// TwinCAT 3 PLC project Transport
// ProgramVersion: 3.1.4026.21
// CompilerDefines: VISU_USEPROPERTYINFO
// libraries:
//   Tc2_Standard, * (Beckhoff Automation GmbH)
//   Tc2_System, * (Beckhoff Automation GmbH)
//   VisuDialogs, * (System)
// project tree:
//   001DUTs/ENUM/ E_CmdState.TcDUT, E_ErrorLevel.TcDUT, E_Mode.TcDUT, E_Convoyer.TcDUT, E_LTUPosition.TcDUT, E_RouteStepType.TcDUT, E_SetChild.TcDUT
//   001DUTs/GVL_Base/ GVL_Core.TcGVL
//   001DUTs/ITF/Device/ ITF_Convoyer.TcIO, ITF_LTU.TcIO, ITF_RouteProvider.TcIO
//   001DUTs/ITF/Generic/ ITF_Base.TcIO, ITF_Device.TcIO
//   001DUTs/ITF/ ITF_Owner.TcIO
//   001DUTs/STRUCT/ ST_ErrorInfo.TcDUT, ST_MaschineHMI.TcDUT, ST_Route.TcDUT, ST_RouteJob.TcDUT, ST_RouteStep.TcDUT
//   002 POUs/00 Generic/ FD_Device.TcPOU, FB_Base.TcPOU, FM_Maschine.TcPOU
//   002 POUs/01 Lib/01 Device/00 Template/ FB_Template.TcPOU (not stored)
//   002 POUs/01 Lib/01 Device/ FD_RouteManagerDevice.TcPOU, FD_LUTDevice.TcPOU (not stored), FD_ConvoyerDevice.TcPOU, FD_RouteExecutorDevice.TcPOU
//   002 POUs/01 Lib/02 SimpleDevice/00 Template/ FB_TemplateSimpleDevice.TcPOU
//   002 POUs/01 Lib/02 SimpleDevice/ FB_ReadHead.TcPOU, FB_PneuCyl_Stopper.TcPOU, FB_SimpleMotor.TcPOU (not stored), FB_PneuCyl_3Pos.TcPOU
//   002 POUs/01 Lib/Digit I_O/Input/ FB_Input.TcPOU (not stored)
//   002 POUs/01 Lib/Digit I_O/Output/ FB_Output.TcPOU
//   1000 Maschine xxx/01 DUTs/GVLs/ GVL_Customer.TcGVL
//   1000 Maschine xxx/01 DUTs/STRUCT/ ST_HmiCustomer.TcDUT
//   1000 Maschine xxx/ MAIN.TcPOU
//   1000 Maschine xxx/_Customer/ FM_Customer.TcPOU
//   1000 Maschine xxx/_Customer/VISUs/ Visu_Customer.TcVIS
//   / GlobalTextList.TcGTLO, PlcTask.TcTTO, Visualisierungsmanager.TcVMO (not stored)
// real-time tasks:
//   TASK PlcTask: cycle T#10ms, priority 20, ADS port 350

CONFIGURATION Transport
    RESOURCE PLC ON TwinCAT3
        TASK PlcTask(INTERVAL := T#10ms, PRIORITY := 20);
        PROGRAM MAIN WITH PlcTask : MAIN;
    END_RESOURCE
END_CONFIGURATION

// ---- 001DUTs/ENUM/E_CmdState.TcDUT

{attribute 'qualified_only'}
{attribute 'strict'}
{attribute 'to_string'}

(*

*)
TYPE E_CmdState :
(
	//====================  
	//											
	Idle							:=  0,
	Succeeded 				:=  1,
	Error	    				:=  2,
	Timeout						:=  3,
	Aborted	    			:=  4,
	Deleted						:=  5,
	Reseted						:=  6,
	NotReady					:=  7,
	Failed						:=  8,
	Hold							:=  9,
	
	//==================== 
	Busy							:= 15
);
END_TYPE

// ---- 001DUTs/ENUM/E_ErrorLevel.TcDUT

{attribute 'qualified_only'}
{attribute 'strict'}
{attribute 'to_string'}
TYPE E_ErrorLevel :
(
	NONE := 0,
	Low,
	High,
	Critical
)UINT;
END_TYPE

// ---- 001DUTs/ENUM/E_Mode.TcDUT
{attribute 'qualified_only'}
{attribute 'strict'}
{attribute 'to_string'}
TYPE E_Mode :
(
 	Idle := 0,
 	Homing,
 	Service,
 	Auto,
 	Error
)UINT;
END_TYPE

// ---- 001DUTs/ENUM/E_Convoyer.TcDUT
{attribute 'qualified_only'}
{attribute 'strict'}
{attribute 'to_string'}
(*

*)
TYPE E_Convoyer :
(
	Convoyer_NONE := 0,
  Convoyer_3		:=3,
  Convoyer_6		:=6,
  Convoyer_9		:=9,
  Convoyer_12		:=12
)UINT;
END_TYPE

// ---- 001DUTs/ENUM/E_LTUPosition.TcDUT
{attribute 'qualified_only'}
{attribute 'strict'}
{attribute 'to_string'}

(*
	Used to define:
	Current LTU position
	Target position (position cible)
	Routing steps
*)

TYPE E_LTUPosition :
(
 	LTU_Unknown := 0,
  LTU_Bottom,
  LTU_Middle,
  LTU_Top
)UINT;
END_TYPE

// ---- 001DUTs/ENUM/E_RouteStepType.TcDUT
{attribute 'qualified_only'}
{attribute 'strict'}
{attribute 'to_string'}
(*
	this ENUM describes elementary actions the system
*)
TYPE E_RouteStepType :
(
 	Route_NONE := 0,

  Route_SetLTUPosition,
  Route_StartConveyor,
  Route_StopConveyor,
  
  Route_StartLTUMotor,
  Route_StopLTUMotor,
  
  Route_WaitLTUOccupied,
  Route_WaitLTUFree,
  Route_WaitLTUPosition,
  
  Route_OpenStopper,
  Route_CloseStopper
)UINT;
END_TYPE

// ---- 001DUTs/ENUM/E_SetChild.TcDUT

{attribute 'qualified_only'}
TYPE E_SetChild :
(
	None					:= 0,
	Enable				:= 1,
	Reset  				:= 3,
	Abort 				:= 4,
	ClearError  	:= 5,
	EStop			  	:= 6,
	Auto  			  := 7,
	Servic				:= 8,
	Home 					:= 9,
	Release		  	:= 10
);
END_TYPE

// ---- 001DUTs/STRUCT/ST_ErrorInfo.TcDUT

TYPE ST_ErrorInfo :
STRUCT
	bActive       : BOOL;
	uiErrorID     : UINT;
	eLevel        : E_ErrorLevel;
	
	sOwner        : STRING(80);
	sMessage      : STRING(255);
	sFullMessage  : STRING(255);
END_STRUCT
END_TYPE

// ---- 001DUTs/STRUCT/ST_MaschineHMI.TcDUT
TYPE ST_MaschineHMI :
STRUCT
	// Commands from HMI
	bCmdHome     					: BOOL;
	bCmdAuto     					: BOOL;
	bCmdService  					: BOOL;
	bCmdStop     					: BOOL;
	bCmdReset    					: BOOL;
	bCmdAbort    					: BOOL;
	
	// Status to HMI
	bEnabled     					: BOOL;
	bReady       					: BOOL;
	bHomed       					: BOOL;
	bBusy        					: BOOL;
	bDone        					: BOOL;
	bError       					: BOOL;
	             					
	eMode        					: E_Mode;
	eCmdState    					: E_CmdState;
	uiSequenceID       		: UINT;
	             					
	sName        					: STRING;
	uiID         					: UINT;
END_STRUCT
END_TYPE

// ---- 001DUTs/STRUCT/ST_Route.TcDUT
(*
This structure contains:
	Source
	Destination
	Number of steps
	Complete routing sequence
*)
TYPE ST_Route :
	STRUCT
  	eSource        : E_Convoyer;
    eDestination   : E_Convoyer;
    iuStepCount    : UINT;
    astSteps       : ARRAY[1..20] OF ST_RouteStep;
	END_STRUCT
END_TYPE

// ---- 001DUTs/STRUCT/ST_RouteJob.TcDUT

TYPE ST_RouteJob :
STRUCT
	uiJobID        	: UINT;
                 	
	eSource        	: E_Convoyer;
	eDestination   	: E_Convoyer;
	               	
	bValid         	: BOOL;
	bReserved      	: BOOL;
	bExecuting     	: BOOL;
	bDone          	: BOOL;
	bError         	: BOOL;
	               	
	stRoute        	: ST_Route;
END_STRUCT
END_TYPE

// ---- 001DUTs/STRUCT/ST_RouteStep.TcDUT
(*
A step represents:
	An action
	On a given transport
	Optionally with an LTU position
*)
TYPE ST_RouteStep :
	STRUCT
		//eStepType      : E_RouteStepType;   // an action
    eConvoyer      : E_Convoyer;				// on a concoyer
    eLTUPosition   : E_LTUPosition;			// an LTU position
	END_STRUCT
END_TYPE

// ---- 1000 Maschine xxx/01 DUTs/STRUCT/ST_HmiCustomer.TcDUT
TYPE ST_HmiCustomer :
STRUCT
	// Commands To PLC
	bCmdHome     					: BOOL;
	bCmdAuto     					: BOOL;
	bCmdService  					: BOOL;
	bCmdStop     					: BOOL;
	bCmdReset    					: BOOL;
	bCmdAbort    					: BOOL;
END_STRUCT
END_TYPE

// ---- 001DUTs/GVL_Base/GVL_Core.TcGVL
{attribute 'qualified_only'}
VAR_GLOBAL CONSTANT
	
C_MaxChild													: UDINT		:=  60;				// maximum number of childs for each device
END_VAR

// ---- 1000 Maschine xxx/01 DUTs/GVLs/GVL_Customer.TcGVL
{attribute 'qualified_only'}
VAR_GLOBAL CONSTANT
	//======================================================= GENARAL 
	
	
	bText    : BOOL :=FALSE ;
	
	//======================================================= Name Device 
	C_Name_fbLutDevice3                : STRING := 'fbLutDevice3';
	C_Name_fbLutDevice6                : STRING := 'fbLutDevice6';
	C_Name_fbLutDevice9                : STRING := 'fbLutDevice9';
	C_Name_fbLutDevice12               : STRING := 'fbLutDevice12';
	
	C_Name_ConvoyerDevice3             : STRING := 'ConvoyerDevice3';
	C_Name_ConvoyerDevice6             : STRING := 'ConvoyerDevice6';
	C_Name_ConvoyerDevice9             : STRING := 'ConvoyerDevice9';
	C_Name_ConvoyerDevice12            : STRING := 'ConvoyerDevice12';
	
	C_Name_RouteManagerDevice          : STRING := 'RouteManagerDevice';

	
	//======================================================= Name Simple Device 
	C_Name_LTUPneuClyZ			           : STRING := 'PneuCylZAxisLTU';
	C_Name_LUTStopper									 : STRING := 'StopperLTU';
	C_Name_LUTDcMotor 						     : STRING := 'LUTSimpleMotor';
	
	C_Name_StopperCarrieConvoyer			 : STRING := 'StopperLTU';
	C_Name_ConvoyerDcMotor						 : STRING := 'StopperLTU';
	C_Name_ReadHead										 : STRING := 'StopperLTU';
	
	
	//======================================================= Name Componemt
	C_Name_LUTLightBarrier 						 : STRING := 'LUTLightBarrier';
	
	C_Name_PneuCylBottomOut 					 : STRING := 'PneuCylBottomOut';
	C_Name_PneuCylTopOut 						   : STRING := 'PneuCylTopOut';
	C_Name_PneuCylBottomIn  					 : STRING := 'PneuCylBottomIn';
	C_Name_PneuCylTopIn 						   : STRING := 'PneuCylTopIn';
	C_Name_PneuCylMiddleIn 						 : STRING := 'PneuCylMiddleIn';
	
	C_Name_DCMotorOut									 : STRING := 'DCMotorOut';
	
	C_Name_StopperOut									 : STRING := 'DCMotorOut';
	C_Name_StopperOccupied						 : STRING := 'DCMotorOut';
	
	
	//======================================================= ID Device 
	//10--99
	C_ID_fbLutDevice3                  : UINT :=  10;
	C_ID_fbLutDevice6                  : UINT :=  11;
	C_ID_fbLutDevice9                  : UINT :=  12;
	C_ID_fbLutDevice12                 : UINT :=  13;
	
	C_ID_ConvoyerDevice3               : UINT :=  14;
	C_ID_ConvoyerDevice6               : UINT :=  15;
	C_ID_ConvoyerDevice9               : UINT :=  16;
	C_ID_ConvoyerDevice12              : UINT :=  17;
	
	C_ID_RouteManagerDevice            : UINT :=  18;
	
	
	//======================================================= Name Simple Device 
	//100--150
	C_ID_LTUPneuClyZ	                 : UINT :=  100;
	C_ID_LUTStopper										 : UINT :=  101;
	C_ID_LUTSimpleMotor								 : UINT :=  101;
	
	C_ID_StopperCarrieConvoyer				 : UINT :=  102;
	C_ID_MotorComvoyer								 : UINT :=  103;
	C_ID_ReadHead       							 : UINT :=  104;
	
	
	//======================================================= Name Componemt
	//
	C_ID_LUTLightBarrier							 : UINT :=  151;
	
	C_ID_PneuCylBottomOut							 : UINT :=  152;
	C_ID_PneuCylTopOut  							 : UINT :=  153;
	
	C_ID_PneuCylBottomIn							 : UINT :=  154;
	C_ID_PneuCylTopIn   							 : UINT :=  155;
	C_ID_PneuCylMiddleIn  						 : UINT :=  156;
	
	C_ID_DCMotorOut										 : UINT :=  157;
	C_ID_StopperOut										 : UINT :=  158;
	C_ID_StopperOccupied							 : UINT :=  159;
	
	
	//======================================================= Customer

	C_Name_Machine                    	: STRING := 'ekvip_Convoyer'; 


	C_ID_Machine                        : UINT :=  200;


 
END_VAR

// ---- 001DUTs/ITF/Device/ITF_Convoyer.TcIO
INTERFACE ITF_Convoyer EXTENDS ITF_Device

PROPERTY CarrierWaiting : BOOL
GET
END_GET
SET
END_SET
END_PROPERTY

PROPERTY Destination : E_Convoyer
GET
END_GET
SET
END_SET
END_PROPERTY

METHOD mCmdExec_TranspOut : E_CmdState
VAR_INPUT
	I_bExecute 			: BOOL;
END_VAR
END_METHOD

PROPERTY RouteGranted : BOOL
GET
END_GET
SET
END_SET
END_PROPERTY

PROPERTY RouteRequest : BOOL
GET
END_GET
SET
END_SET
END_PROPERTY

PROPERTY Source : E_Convoyer
GET
END_GET
SET
END_SET
END_PROPERTY

PROPERTY TranspOutBusy : BOOL
GET
END_GET
SET
END_SET
END_PROPERTY

PROPERTY TranspOutDone : BOOL
GET
END_GET
SET
END_SET
END_PROPERTY

PROPERTY TranspOutRequest : BOOL
GET
END_GET
SET
END_SET
END_PROPERTY

END_INTERFACE

// ---- 001DUTs/ITF/Device/ITF_LTU.TcIO
INTERFACE ITF_LTU EXTENDS ITF_Device

PROPERTY CarrierPresent : BOOL
GET
END_GET
SET
END_SET
END_PROPERTY

PROPERTY LTUFree : BOOL
GET
END_GET
SET
END_SET
END_PROPERTY

PROPERTY LTUPosition : E_LTUPosition
GET
END_GET
SET
END_SET
END_PROPERTY

METHOD mCmdExec_MoveMiddle : E_CmdState
VAR_INPUT
	I_bExecute					: BOOL;
END_VAR
END_METHOD

METHOD mCmdExec_MoveTop : E_CmdState
VAR_INPUT
	I_bExecute					: BOOL;
END_VAR
END_METHOD

METHOD mCmdExec_TransferTop : E_CmdState
VAR_INPUT
	I_bExecute					: BOOL;
END_VAR
END_METHOD

METHOD mGetLTUByConvoyer : E_CmdState
VAR_INPUT
	I_bExecute					: BOOL;
END_VAR
END_METHOD

PROPERTY ReservedBy : E_Convoyer
GET
END_GET
SET
END_SET
END_PROPERTY

END_INTERFACE

// ---- 001DUTs/ITF/Device/ITF_RouteProvider.TcIO
INTERFACE ITF_RouteProvider

METHOD mGetNextRoute : E_CmdState
VAR_OUTPUT
	O_pRouteJob				: POINTER TO ST_RouteJob;
END_VAR
END_METHOD

METHOD mReleaseRoute : E_CmdState
VAR_INPUT
	I_uiJobID					 : UINT;
END_VAR
END_METHOD

END_INTERFACE

// ---- 001DUTs/ITF/Generic/ITF_Base.TcIO
INTERFACE ITF_Base EXTENDS __System.IQueryInterface

PROPERTY Busy : BOOL
GET
END_GET
SET
END_SET
END_PROPERTY

PROPERTY Done : BOOL
GET
END_GET
SET
END_SET
END_PROPERTY

PROPERTY Enable : BOOL
GET
END_GET
SET
END_SET
END_PROPERTY

PROPERTY Error : BOOL
GET
END_GET
SET
END_SET
END_PROPERTY

PROPERTY ErrorID : UINT
GET
END_GET
SET
END_SET
END_PROPERTY

PROPERTY ErrorLevel : E_ErrorLevel
GET
END_GET
SET
END_SET
END_PROPERTY

PROPERTY ErrorMessage : STRING
GET
END_GET
SET
END_SET
END_PROPERTY

PROPERTY ErrorOwner : STRING
GET
END_GET
SET
END_SET
END_PROPERTY

PROPERTY ID : UINT
GET
END_GET
SET
END_SET
END_PROPERTY

METHOD mClearError : BOOL
VAR_INPUT
END_VAR
END_METHOD

METHOD mEnable : bool
VAR_INPUT
END_VAR
END_METHOD

METHOD mError : BOOL
VAR_INPUT
	I_sMessage   : STRING;
	I_eLevel		 : E_ErrorLevel;
	I_uiError		 : UINT;
END_VAR
END_METHOD

METHOD mInit : bool
VAR_INPUT

END_VAR
END_METHOD

METHOD mReset : BOOL
VAR_INPUT
	
END_VAR
END_METHOD

PROPERTY Name : STRING
GET
END_GET
SET
END_SET
END_PROPERTY

END_INTERFACE

// ---- 001DUTs/ITF/Generic/ITF_Device.TcIO
INTERFACE ITF_Device EXTENDS ITF_BASE

PROPERTY Homed : BOOL
GET
END_GET
SET
END_SET
END_PROPERTY

METHOD mAbort : E_CmdState
VAR_INPUT
	I_bExecute : BOOL;
END_VAR
END_METHOD

METHOD mAutomatic : E_CmdState
VAR_INPUT
	I_bExecute : BOOL;
END_VAR
END_METHOD

METHOD mDone : E_CmdState
VAR_INPUT
END_VAR
END_METHOD

METHOD mHold : E_CmdState
VAR_INPUT
	I_bExecute : BOOL;
END_VAR
END_METHOD

METHOD mHome : E_CmdState
VAR_INPUT
	I_bExecute : BOOL;
END_VAR
END_METHOD

PROPERTY Mode : E_Mode
GET
END_GET
SET
END_SET
END_PROPERTY

METHOD mRelease : E_CmdState
VAR_INPUT
	I_bExecute : BOOL;
END_VAR
END_METHOD

METHOD mSequence : E_CmdState
VAR_INPUT
	I_bExecute : BOOL;
END_VAR
END_METHOD

METHOD mService : E_CmdState
VAR_INPUT
	I_bExecute : BOOL;
END_VAR
END_METHOD

METHOD mStop : E_CmdState
VAR_INPUT
	I_bExecute : BOOL;
END_VAR
END_METHOD

PROPERTY Ready : BOOL
GET
END_GET
SET
END_SET
END_PROPERTY

PROPERTY SequenceBusy : BOOL
GET
END_GET
SET
END_SET
END_PROPERTY

PROPERTY SequenceDone : BOOL
GET
END_GET
SET
END_SET
END_PROPERTY

END_INTERFACE

// ---- 001DUTs/ITF/ITF_Owner.TcIO
INTERFACE ITF_Owner EXTENDS __System.IQueryInterface

METHOD mRegisterChild : BOOL
VAR_INPUT
	I_itfChild  : ITF_Device;
END_VAR
END_METHOD

END_INTERFACE

// ---- 1000 Maschine xxx/MAIN.TcPOU
PROGRAM MAIN
VAR
	fbCustomer										: FM_Customer( GVL_Customer.C_Name_Machine,
																							 GVL_Customer.C_ID_Machine,
																						   NULL,
																							);
END_VAR


fbCustomer();

END_PROGRAM

// ---- 1000 Maschine xxx/_Customer/FM_Customer.TcPOU
FUNCTION_BLOCK FM_Customer EXTENDS FM_Maschine
VAR_INPUT
END_VAR
VAR_OUTPUT
END_VAR
VAR
	// ===============================
	stHMI 														: ST_MaschineHMI;
	
	// =============================== Instance
	
	fdLUTDevice3											: FD_LUTDevice 					(GVL_Customer.C_Name_fbLutDevice3,  // Name
																								   					GVL_Customer.C_ID_fbLutDevice3,		  // ID
																								   					THIS^,															// ITF_Owner
																								   					);
																								   					
	fdLUTDevice6											: FD_LUTDevice 					(GVL_Customer.C_Name_fbLutDevice6,  // Name
																								   					GVL_Customer.C_ID_fbLutDevice6,		  // ID
																								   					THIS^,															// ITF_Owner
																								   					);
                    		  					               					
	fdLUTDevice9											: FD_LUTDevice 					(GVL_Customer.C_Name_fbLutDevice9,  // Name
																								   					GVL_Customer.C_ID_fbLutDevice9,		  // ID
																								   					THIS^,															// ITF_Owner
																								   					);
																							          		
	fdLUTDevice12			      					: FD_LUTDevice					(GVL_Customer.C_Name_fbLutDevice12,  // Name
																														GVL_Customer.C_ID_fbLutDevice12,		 // ID
																														THIS^,															 // ITF_Owner
																														);
																														
	fdConvoyerDevice3			  					: FD_ConvoyerDevice			(GVL_Customer.C_Name_ConvoyerDevice3,  // Name
																						 				      	GVL_Customer.C_ID_ConvoyerDevice3,		 // ID
																										    		THIS^,															  // ITF_Owner
																														E_Convoyer.Convoyer_3,								// Source ID
																										      	);
																														
	fdConvoyerDevice6			  					: FD_ConvoyerDevice			(GVL_Customer.C_Name_ConvoyerDevice6,  // Name
																						 				      	GVL_Customer.C_ID_ConvoyerDevice6,		 // ID
																										    		THIS^,															   // ITF_Owner
																														E_Convoyer.Convoyer_6,								// Source ID
																										      	);
                                                          	
	fdConvoyerDevice9			  					: FD_ConvoyerDevice			(GVL_Customer.C_Name_ConvoyerDevice9,  // Name
																						 				      	GVL_Customer.C_ID_ConvoyerDevice9,		 // ID
																										    		THIS^,															   // ITF_Owner
																														E_Convoyer.Convoyer_9,								// Source ID
																										      	);
                                                          	
	fdConvoyerDevice12			  			  : FD_ConvoyerDevice		  (GVL_Customer.C_Name_ConvoyerDevice12,  // Name
																						 				        GVL_Customer.C_ID_ConvoyerDevice12,		  // ID
																										    	  THIS^,															    // ITF_Owner
																														E_Convoyer.Convoyer_12,								// Source ID
																										        );																										
			
	fdRouteManager			  						: FD_RouteManagerDevice		  (GVL_Customer.C_Name_RouteManagerDevice,   // Name
																						 				        GVL_Customer.C_ID_RouteManagerDevice,		 // ID
																										    	  THIS^,															     // ITF_Owner
																														fdLUTDevice3,   												 //ITF_LTUDevice
																														fdLUTDevice6,	 													 //ITF_LTUDevice
																														fdLUTDevice9,	 													 //ITF_LTUDevice
																														fdLUTDevice12,	 												 //ITF_LTUDevice
																														fdConvoyerDevice3,                       // ITF_Convoyer
																														fdConvoyerDevice6,                       // ITF_Convoyer
																														fdConvoyerDevice9,                       // ITF_Convoyer
																														fdConvoyerDevice12,                      // ITF_Convoyer
																										      );
																													
	fdRouteExecutorDevice			  			: FD_RouteExecutorDevice		  (GVL_Customer.C_Name_RouteManagerDevice,   // Name
																						 				        				GVL_Customer.C_ID_RouteManagerDevice,		 // ID
																										    	  				THIS^,															     // ITF_Owner
																																		fdLUTDevice3,   												 //ITF_LTUDevice
																																		fdLUTDevice6,	 													 //ITF_LTUDevice
																																		fdLUTDevice9,	 													 //ITF_LTUDevice
																																		fdLUTDevice12,	 												 //ITF_LTUDevice
																																		fdConvoyerDevice3,                       // ITF_Convoyer
																																		fdConvoyerDevice6,                       // ITF_Convoyer
																																		fdConvoyerDevice9,                       // ITF_Convoyer
																																		fdConvoyerDevice12,                      // ITF_Convoyer
																																		fdRouteManager,
																										      				);																													
																				
END_VAR


//must !! 
SUPER^();  
//====================================
IF NOT Enable THEN RETURN; END_IF
//HMI
mVisu();

//Device instance
fdLUTDevice3();
fdLUTDevice6();
fdLUTDevice9();
fdLUTDevice12();

fdConvoyerDevice3();
fdConvoyerDevice6();
fdConvoyerDevice9();
fdConvoyerDevice12();

fdRouteManager();
fdRouteExecutorDevice();

//FB_Init ist immer implizit verfügbar und wird primär für die Initialisierung verwendet.
//Der Rückgabewert wird nicht ausgewertet. Für gezielte Einflussnahme können Sie
//die Methoden explizit deklarieren und darin mit dem Standard-Initialisierungscode 
//zusätzlichen Code bereitstellen. Sie können den Rückgabewert auswerten.
METHOD FB_Init: BOOL
VAR_INPUT    
	bInitRetains					: BOOL; 					// TRUE: Die Retain-Variablen werden initialisiert (Reset warm / Reset kalt)    
	bInCopyCode						: BOOL;  					// TRUE: Die Instanz wird danach in den Kopiercode kopiert (Online-Change)
	
	I_Name                : STRING;         //  Name
	I_ID                  : UINT;           // ID
  I_itfOwner					  : ITF_Owner;      // owner 
END_VAR
END_METHOD

METHOD mVisu : BOOL
VAR_INPUT
	
END_VAR
super^.mVisu();

// Machine status -->HMI
//==================================================

stHMI.bReady 								:= Ready;
stHMI.bBusy  								:= SequenceBusy;
stHMI.bDone  								:= SequenceDone;
stHMI.bError 								:= Error;
stHMI.bHomed 								:= Homed;

stHMI.eMode 								:= Mode;

stHMI.uiSequenceID 					:= SequenceID;

// HMI commands
//==================================================

//------------------------------
// HOME
IF stHMI.bCmdHome 
	THEN
  	stHMI.eCmdState 				:= mHome(TRUE);
    stHMI.bCmdHome 					:= FALSE;
END_IF

//------------------------------
// AUTO
IF stHMI.bCmdAuto 
	THEN
  	stHMI.eCmdState 				:= mAutomatic(TRUE);
    stHMI.bCmdAuto 					:= FALSE;
END_IF

//------------------------------
// SERVICE
IF stHMI.bCmdService 
	THEN
    stHMI.eCmdState 				:= mService( TRUE);
    stHMI.bCmdService 			:= FALSE;
END_IF

//------------------------------
// STOP
IF stHMI.bCmdStop 
	THEN
    stHMI.eCmdState 				:= mStop(TRUE);
    stHMI.bCmdStop 					:= FALSE;
END_IF

//------------------------------
// ABORT

IF stHMI.bCmdAbort 
	THEN
    stHMI.eCmdState := mAbort(TRUE);
    stHMI.bCmdAbort := FALSE;
END_IF

//------------------------------
// RESET
IF stHMI.bCmdReset 
	THEN
  	mReset();
    stHMI.bCmdReset := FALSE;
END_IF
//=========================================================
mVisu := TRUE;
END_METHOD

END_FUNCTION_BLOCK

// ---- 002 POUs/00 Generic/FM_Maschine.TcPOU
FUNCTION_BLOCK ABSTRACT FM_Maschine EXTENDS FD_Device 
VAR_INPUT
END_VAR
VAR_OUTPUT
END_VAR
VAR
	// Global child status
	bAllChildsReady 					: BOOL;
	bAllChildsHomed 					: BOOL;
	bAllChildsDone  					: BOOL;
	bAnyChildBusy   					: BOOL;
	bAnyChildError  					: BOOL;
	// Internal command state
	//eLastChildCmdState 				: E_CmdState;
	
	// Hmi Variable
END_VAR


SUPER^();  
IF NOT Enable THEN RETURN; END_IF;

// Update global child status every PLC cycle
mUpdateChildsState();

IF SequenceBusy THEN
    mSequence(TRUE);
END_IF

//FB_Init ist immer implizit verfügbar und wird primär für die Initialisierung verwendet.
//Der Rückgabewert wird nicht ausgewertet. Für gezielte Einflussnahme können Sie
//die Methoden explizit deklarieren und darin mit dem Standard-Initialisierungscode 
//zusätzlichen Code bereitstellen. Sie können den Rückgabewert auswerten.
METHOD FB_Init: BOOL
VAR_INPUT    
	bInitRetains					: BOOL; 					// TRUE: Die Retain-Variablen werden initialisiert (Reset warm / Reset kalt)    
	bInCopyCode						: BOOL;  					// TRUE: Die Instanz wird danach in den Kopiercode kopiert (Online-Change)
	
	I_Name                : STRING;         //  Name
	I_ID                  : UINT;           // ID
  I_itfOwner					  : ITF_Owner;      // owner 
END_VAR

	bConfigurationBasePos := FALSE;
	bAnyChildBusy   			:= FALSE;
	bAnyChildError  			:= FALSE;
	bAllChildsReady 			:= TRUE;
	bAllChildsHomed 			:= TRUE;
	bAllChildsDone  			:= TRUE;
END_METHOD

METHOD mAutomatic : E_CmdState
VAR_INPUT
	I_bExecute	: BOOL;
END_VAR

VAR_INST
	bYann  	: BOOL;
	bYann2  	: BOOL;
	
END_VAR

IF bYann 
	THEN
	bYann2 := true;
END_IF
bAllChildsHomed	:= TRUE;
// Call mAutomatic in Base
mAutomatic := SUPER^.mAutomatic(I_bExecute);

// Machine can only go AUTO if all child devices are homed
mUpdateChildsState();

IF NOT bAllChildsHomed 
	THEN
    mAutomatic := E_CmdState.NotReady;
    RETURN;
END_IF
END_METHOD

METHOD mCheckAllChildsReady : Bool
VAR_INPUT
END_VAR
END_METHOD

METHOD mHome : E_CmdState
VAR_INPUT
	I_bExecute	: BOOL;
END_VAR

mHome := SUPER^.mHome(I_bExecute);

// If generic checks failed -> exit
IF (mHome <> E_CmdState.Busy) AND NOT ConfigurationBasePos THEN RETURN; END_IF

// Machine-specific preparation
mUpdateChildsState();

// verify children available before homing
IF bAnyChildError 
	THEN
    mHome := E_CmdState.Error;
    RETURN;
END_IF
END_METHOD

METHOD mReset : BOOL
VAR_INPUT
END_VAR
VAR
	L_uiIndex   : UINT;
END_VAR

// Reset own machine state from parent class
//==================================================
SUPER^.mReset();

// Reset all register child devices
//==================================================
FOR L_uiIndex := 1 TO uiChildsCount DO
	aitfChilds[L_uiIndex].mReset();
END_FOR

// Reset machine supervision flags
//==================================================
bAllChildsReady 							:= FALSE;
bAllChildsHomed 							:= FALSE;
bAllChildsDone  							:= FALSE;
                							
bAnyChildBusy   							:= FALSE;
bAnyChildError  							:= FALSE;

// Reset machine sequence
//==================================================
SequenceID 										:= C_SeqStep_Idle;
              								
bSequenceBusy 								:= FALSE;
bSequenceDone 								:= FALSE;
              								
bReady 												:= FALSE;
bHomed 												:= FALSE;

// Reset machine mode
//==================================================
Mode 													:= E_Mode.IDLE;

// Reset successful
//==================================================
mReset := TRUE;
END_METHOD

METHOD mSequence : E_CmdState
VAR_INPUT
	I_bExecute				: BOOL;
END_VAR

VAR
    eCmd 						: E_CmdState;
END_VAR

// Generic pre-check from parent
mSequence := SUPER^.mSequence(I_bExecute := I_bExecute);

IF mSequence <> E_CmdState.Busy THEN
    RETURN;
END_IF

// Update child status before sequence logic
mUpdateChildsState();

IF bAnyChildError THEN
    SequenceID := C_SeqStep_Error;
END_IF

CASE SequenceID OF
	C_SeqStep_Idle:
		;
	C_SeqStep_Start:
	    CASE Mode OF
	    	E_Mode.Homing:
	    	    eCmd 	:= mSetChildMode(E_Mode.Homing);
	    	E_Mode.Auto:
	    	    eCmd 	:= mSetChildMode(E_Mode.Auto);
	    	E_Mode.Service:
	    	    eCmd 	:= mSetChildMode(E_Mode.Service);
	    END_CASE
		SequenceID  := C_SeqStep_Running;
	  mSequence 	:= E_CmdState.Busy;
	 
	C_SeqStep_Running:
	    // Wait until all child devices finish their requested command
	    mUpdateChildsState();
	 
	    IF bAnyChildError THEN
	        SequenceID := C_SeqStep_Error;
	 
	    ELSIF NOT bAnyChildBusy THEN
	        SequenceID := C_SeqStep_Done;
	    END_IF
	    mSequence := E_CmdState.Busy;
		
	C_SeqStep_Done:
		bSequenceBusy := FALSE;
		bSequenceDone := TRUE;
		
		IF Mode = E_Mode.Homing 
	  	THEN
		    bHomed := TRUE;
		END_IF
		
		bReady := TRUE;
		SequenceID := C_SeqStep_Idle;
		
		mSequence := E_CmdState.Succeeded;
		
	C_SeqStep_Error:
		bError 				:= TRUE;
		bSequenceBusy := FALSE;
		bSequenceDone := FALSE;
		
		mSequence := E_CmdState.Error;
		
	ELSE
		SequenceID := C_SeqStep_Error;
		mSequence := E_CmdState.Error;
END_CASE
END_METHOD

METHOD mService : E_CmdState
VAR_INPUT
	I_bExecute : BOOL;
END_VAR
IF NOT I_bExecute 
	THEN
    mService := E_CmdState.Idle;
    RETURN;
END_IF

Mode := E_Mode.Service;
bSequenceBusy := FALSE;
bSequenceDone := FALSE;

mService := E_CmdState.Busy;
END_METHOD

METHOD PROTECTED mSetChildMode  : E_CmdState
VAR_INPUT
	I_eMode 		: E_Mode;
END_VAR

VAR
	uiIndex 		: UINT;
  eCmd 				: E_CmdState;
END_VAR

mSetChildMode := E_CmdState.Succeeded;

// Send requested mode command to all child devices
FOR uiIndex := 1 TO uiChildsCount DO
	CASE I_eMode OF
  	E_Mode.Homing:
  		eCmd 			    := aitfChilds[uiIndex].mHome(TRUE);
  	E_Mode.Auto:
  		eCmd 			    := aitfChilds[uiIndex].mAutomatic(TRUE);
  	E_Mode.Service:
  		eCmd 			    := aitfChilds[uiIndex].mService(TRUE);			
		E_Mode.Idle:
  		eCmd 			    := aitfChilds[uiIndex].mStop(TRUE);
  	E_Mode.Error:
  		eCmd 			    := aitfChilds[uiIndex].mAbort(TRUE);
  END_CASE

  // If one child is busy, global command is still busy
	IF eCmd = E_CmdState.Busy 
		THEN
	    mSetChildMode  := E_CmdState.Busy;
	END_IF
	 
	// If one child has error, global command is error
	IF (eCmd = E_CmdState.Error) OR (eCmd = E_CmdState.NotReady) 
  	THEN
	    mSetChildMode  := eCmd;
	    RETURN;
	END_IF
END_FOR
END_METHOD

METHOD mStop : E_CmdState
VAR_INPUT
	I_bExecute	: BOOL;
END_VAR

// Stop machine base status
SUPER^.mStop(I_bExecute);

// Stop all child devices
 //StopChilds();
END_METHOD

METHOD PROTECTED mStopChilds  : E_CmdState
VAR_INPUT
END_VAR

VAR
    uiIndex 				: UINT;
    eCmd 						: E_CmdState;
END_VAR

mStopChilds := E_CmdState.Succeeded;

// Stop all child devices
FOR uiIndex := 1 TO uiChildsCount DO
	eCmd := aitfChilds[uiIndex].mStop(TRUE);
	
	IF eCmd = E_CmdState.Busy 
		THEN
	    mStopChilds := E_CmdState.Busy;
	END_IF
	
	IF eCmd = E_CmdState.Error 
		THEN
	    mStopChilds := E_CmdState.Error;
	    RETURN;
    END_IF
END_FOR
END_METHOD

METHOD PROTECTED mUpdateChildsState  : BOOL
VAR_INPUT
END_VAR
VAR
	L_uiIndex									: UINT;
	
END_VAR

// Evaluate all registered child devices
FOR L_uiIndex := 1 TO uiChildsCount DO

    IF aitfChilds[L_uiIndex].Error THEN
        bAnyChildError := TRUE;
    END_IF

    IF aitfChilds[L_uiIndex].SequenceBusy THEN
        bAnyChildBusy := TRUE;
    END_IF

    IF NOT aitfChilds[L_uiIndex].Ready THEN
        bAllChildsReady := FALSE;
    END_IF

    IF NOT aitfChilds[L_uiIndex].Homed THEN
        bAllChildsHomed := FALSE;
    END_IF

    IF NOT aitfChilds[L_uiIndex].SequenceDone THEN
        bAllChildsDone := FALSE;
    END_IF

END_FOR

mUpdateChildsState := TRUE;
END_METHOD

END_FUNCTION_BLOCK

// ---- 002 POUs/00 Generic/FD_Device.TcPOU
(*
Purpose:     Base for Devices 
             FD_Device includes standard properties and standard methodes
*)

FUNCTION_BLOCK ABSTRACT FD_Device EXTENDS FB_Base IMPLEMENTS ITF_Device, ITF_Owner
VAR_INPUT
END_VAR
VAR_OUTPUT
END_VAR
VAR
	itfDeviceRegister									: ITF_Owner;
	aitfChilds												: ARRAY [1..GVL_Core.C_MaxChild] OF ITF_Device;     // Registered child devices
	uiChildsCount											: UINT := 0;                                       	// Number of registered child devices
	
	eMode															: E_Mode;
	uiSequenceID          						: UINT;
	uiNextStep      									: UINT;
	
	bConfigurationBasePos 						: BOOL;               									
	bHomed          									: BOOL;
	bReady          									: BOOL;
	                									
	bSequenceBusy   									: BOOL;
	bSequenceDone   									: BOOL;
	                									
	bHold           									: BOOL;
	bAbort          									: BOOL;

END_Var

VAR CONSTANT
 //***********************************************************  CONSTANT  C_SeqStep
 C_SeqStep_Idle                   	: UINT :=	0;                    
 C_SeqStep_Start                  	: UINT :=	1; 
 C_SeqStep_Running                  : UINT :=	2;			              
 C_SeqStep_Error                		: UINT :=	3;  									
 C_SeqStep_Abort                		: UINT :=	4;  									 
 C_SeqStep_Undefined            		: UINT :=	5;  							
 C_SeqStep_Done                 		: UINT :=	6;
	
END_VAR


SUPER^();
IF NOT Enable THEN RETURN; END_IF;

IF bError
	THEN
  	mStop(TRUE);
    RETURN;
END_IF;

IF bSequenceBusy THEN mSequence(TRUE); END_IF;

PROPERTY ConfigurationBasePos : BOOL
GET
ConfigurationBasePos := bConfigurationBasePos;
END_GET
SET
bConfigurationBasePos := ConfigurationBasePos;
END_SET
END_PROPERTY

//FB_Init ist immer implizit verfügbar und wird primär für die Initialisierung verwendet.
//Der Rückgabewert wird nicht ausgewertet. Für gezielte Einflussnahme können Sie
//die Methoden explizit deklarieren und darin mit dem Standard-Initialisierungscode 
//zusätzlichen Code bereitstellen. Sie können den Rückgabewert auswerten.
METHOD FB_Init: BOOL
VAR_INPUT    
	bInitRetains					: BOOL; 					// TRUE: Die Retain-Variablen werden initialisiert (Reset warm / Reset kalt)    
	bInCopyCode						: BOOL;  					// TRUE: Die Instanz wird danach in den Kopiercode kopiert (Online-Change)
	
	I_Name                : STRING;         //  Name
	I_ID                  : UINT;           // ID
  I_itfOwner					  : ITF_Owner;      // owner 
END_VAR

IF I_itfOwner <>0
	THEN
		itfDeviceRegister 	:= I_itfOwner;
		itfDeviceRegister.mRegisterChild(THIS^);
END_IF

// Default sequence state
SequenceID 							:= C_SeqStep_Idle;

bSequenceBusy 					:= FALSE;
bSequenceDone 					:= FALSE;
              					
bReady 									:= FALSE;
bHomed									:= FALSE;
bAbort 									:= FALSE;
bHold 									:= FALSE;

bConfigurationBasePos   := TRUE; // provisorisch.
END_METHOD

PROPERTY Homed : BOOL
GET
Homed := bHomed;
END_GET
SET
bHomed := Homed;
END_SET
END_PROPERTY

METHOD mAbort : E_CmdState
VAR_INPUT
	I_bExecute : BOOL;
END_VAR
IF NOT I_bExecute 
	THEN
    mAbort     := E_CmdState.Idle;
    RETURN;
END_IF

bAbort         := TRUE;
bSequenceBusy  := FALSE;
bSequenceDone  := FALSE;

SequenceID     := C_SeqStep_Idle;

mStop(TRUE);

mAbort := E_CmdState.Busy;
END_METHOD

METHOD mAutomatic: E_CmdState
VAR_INPUT
	I_bExecute : BOOL;
END_VAR
// No command requested.
IF NOT I_bExecute THEN
    mAutomatic := E_CmdState.Idle;
    RETURN;
END_IF

// Device disabled / not initialized / not homming
IF NOT Enable OR NOT bHomed
	THEN
    mAutomatic := E_CmdState.NotReady;
    RETURN;
END_IF

// Device is in error state.
IF bError 
	THEN
		SequenceID := C_SeqStep_Error;
    mAutomatic := E_CmdState.Error;
    RETURN;
END_IF

Mode := E_Mode.Auto;

// Start sequence execution.
bSequenceBusy 	:= TRUE;
bSequenceDone 	:= FALSE;
SequenceID     	:= C_SeqStep_Start;
mAutomatic 			:= E_CmdState.Busy;
END_METHOD

METHOD mDone : E_CmdState
VAR_INPUT
END_VAR
(*


*)
IF bError
  THEN 
		mDone :=  E_CmdState.Failed;	
  ELSE 
		mDone :=  E_CmdState.Succeeded;
END_IF

bSequenceBusy := FALSE;
bSequenceDone := TRUE;
SequenceID := C_SeqStep_Idle;
END_METHOD

METHOD mHold : E_CmdState
VAR_INPUT
	I_bExecute : BOOL;
END_VAR

IF NOT I_bExecute 
	THEN
    mHold := E_CmdState.Idle;
    RETURN;
END_IF

bHold := TRUE;
bSequenceBusy := FALSE;
mHold := E_CmdState.Hold;
END_METHOD

METHOD mHome : E_CmdState
VAR_INPUT
	I_bExecute : BOOL;
END_VAR
// No command requested.
IF NOT I_bExecute 
	THEN
    mHome := E_CmdState.Idle;
    RETURN;
END_IF

// Device disabled.
IF NOT Enable 
	THEN
    mHome := E_CmdState.NotReady;
    RETURN;
END_IF

// Device in error.
IF Error 
	THEN
    mHome := E_CmdState.Error;
    RETURN;
END_IF
// Device already running another sequence
IF SequenceBusy 
	THEN
    mHome := E_CmdState.Busy;
    RETURN;
END_IF

// No base position required
// Device is considered homed immediately
IF ConfigurationBasePos 
	THEN
    Mode := E_Mode.Homing;

    Homed := TRUE;
    Ready := TRUE;

    SequenceBusy := FALSE;
    SequenceDone := TRUE;
    SequenceID := C_SeqStep_Idle;

    mHome := E_CmdState.Succeeded;
    RETURN;
END_IF

// Start local homing sequence
Mode := E_Mode.Homing;

SequenceBusy := TRUE;
SequenceDone := FALSE;

Homed := FALSE;
Ready := FALSE;

SequenceID := C_SeqStep_Start;

mHome := E_CmdState.Busy;
END_METHOD

PROPERTY Mode : E_Mode
GET
Mode := eMode;
END_GET
SET
eMode := Mode;
END_SET
END_PROPERTY

METHOD mRegisterChild : BOOL			 
VAR_INPUT
	I_itfChild        : ITF_Device;
END_VAR

VAR 
	L_Itf_ChildDevice : ITF_Device := 0;
END_VAR

IF __QUERYINTERFACE (I_itfChild, L_Itf_ChildDevice)
	THEN 
		IF uiChildsCount < GVL_Core.C_MaxChild
			THEN 
				uiChildsCount 								:= uiChildsCount +1;	
				aitfChilds[uiChildsCount] 		:= L_Itf_ChildDevice;
		END_IF
END_IF
END_METHOD

METHOD mRelease : E_CmdState
VAR_INPUT
	I_bExecute : BOOL;
END_VAR

IF NOT I_bExecute 
	THEN
    mRelease 	:= E_CmdState.Idle;
    RETURN;
END_IF

bHold    			:= FALSE;
bAbort   			:= FALSE;
         			
mRelease 			:= E_CmdState.Busy;
END_METHOD

METHOD mReset : BOOL
VAR_INPUT

END_VAR

SUPER^.mReset();

SequenceID := C_SeqStep_Idle;
END_METHOD

METHOD mSequence : E_CmdState
VAR_INPUT
	I_bExecute : BOOL;
END_VAR

IF NOT I_bExecute 
	THEN
    mSequence := E_CmdState.Idle;
    RETURN;
END_IF

IF bError 
	THEN
		SequenceID := C_SeqStep_Error;
    mSequence  := E_CmdState.Error;
    RETURN;
END_IF

// Allows for a clean stop of a sequence
IF bAbort 
	THEN
    SequenceID := C_SeqStep_Abort;
    mSequence := E_CmdState.Aborted;
    RETURN;
END_IF

//Hold allows for pausing without losing the SequenceID.
IF bHold 
	THEN
    mSequence := E_CmdState.Busy;
    RETURN;
END_IF

bSequenceBusy := TRUE;
bSequenceDone := FALSE;

mSequence := E_CmdState.Busy;
END_METHOD

METHOD mService : E_CmdState
VAR_INPUT
	I_bExecute : BOOL;
END_VAR
IF NOT I_bExecute 
	THEN
    mService := E_CmdState.Idle;
    RETURN;
END_IF

Mode := E_Mode.Service;
bSequenceBusy := FALSE;
bSequenceDone := FALSE;

mService := E_CmdState.Busy;
END_METHOD

METHOD mSetChildOpMode : BOOL
VAR_INPUT
	I_eSetChilds  : E_SetChild;
END_VAR
VAR
	L_uiIndex			: UINT;
END_VAR

FOR L_uiIndex := 1 TO uiChildsCount DO
	CASE I_eSetChilds OF
		E_SetChild.None					: ;
		E_SetChild.Enable				:	aitfChilds[L_uiIndex].Enable:= Enable; 
		E_SetChild.Reset 				: aitfChilds[L_uiIndex].mReset();	
		E_SetChild.Abort				:	aitfChilds[L_uiIndex].mAbort(TRUE);
//		E_SetChild.ClearError		:	aitfChilds[L_uiIndex].mError(TRUE);
		E_SetChild.EStop				:	aitfChilds[L_uiIndex].mStop(TRUE);
		E_SetChild.Auto					: aitfChilds[L_uiIndex].mAutomatic(TRUE);
		E_SetChild.Servic				: aitfChilds[L_uiIndex].mService(TRUE);
		E_SetChild.Home					: aitfChilds[L_uiIndex].mHome(TRUE);
		E_SetChild.Release			: aitfChilds[L_uiIndex].mRelease(TRUE);
	END_CASE
END_FOR
END_METHOD

METHOD mStop : E_CmdState
VAR_INPUT
	I_bExecute : BOOL;
END_VAR
IF NOT I_bExecute 
	THEN
  	mStop 			:= E_CmdState.Idle;
    RETURN;
END_IF

Mode := E_Mode.Error;

bBusy 					:= FALSE;
bDone 					:= FALSE;
bSequenceBusy 	:= FALSE;
bSequenceDone 	:= FALSE;

SequenceID     	:= C_SeqStep_Idle;
mStop 					:= E_CmdState.Succeeded;
END_METHOD

PROPERTY Ready : BOOL
GET
Ready := bReady;
END_GET
SET
bReady := Ready;
END_SET
END_PROPERTY

PROPERTY SequenceBusy : BOOL
GET
SequenceBusy := bSequenceBusy;
END_GET
SET
bSequenceBusy := SequenceBusy;
END_SET
END_PROPERTY

PROPERTY SequenceDone : BOOL
GET
SequenceDone := bSequenceDone ;
END_GET
SET
bSequenceDone := SequenceDone ;
END_SET
END_PROPERTY

PROPERTY SequenceID : UINT
GET
SequenceID := uiSequenceID;
END_GET
SET
uiSequenceID := SequenceID;
END_SET
END_PROPERTY

END_FUNCTION_BLOCK

// ---- 002 POUs/00 Generic/FB_Base.TcPOU
FUNCTION_BLOCK ABSTRACT FB_Base IMPLEMENTS ITF_Base

VAR
	sName          										: STRING;
	uiId           										: UINT;
	
	              										
	bEnable        										: BOOL := TRUE;
	bInit          										: BOOL;
	bBusy          										: BOOL;
	bDone          										: BOOL;
	
	stError 													: ST_ErrorInfo;
	bError         										: BOOL;
	eErrorLevel												: E_ErrorLevel;
	uiErrorID													: UINT;
	sErrorOwner												: STRING;
	sErrorMessage  										: STRING;
END_VAR


IF NOT Init
  THEN Init := mInit();
END_IF

mVisu();

Enable := Enable;
IF NOT Enable 
	THEN 
		bBusy := FALSE;
		bDone := FALSE;
		RETURN; 
END_IF

mEnable();

PROPERTY Busy : bool
GET
Busy := bBusy;
END_GET
SET
bBusy := Busy;
END_SET
END_PROPERTY

PROPERTY Done : bool
GET
Done := bDone;
END_GET
SET
bDone := Done;
END_SET
END_PROPERTY

PROPERTY Enable : BOOL
GET
Enable := bEnable;
END_GET
SET
bEnable := Enable;
END_SET
END_PROPERTY

PROPERTY Error : bool
GET
Error := bError;
END_GET
SET
bError := Error;
END_SET
END_PROPERTY

PROPERTY ErrorID : UINT
GET
ErrorID := uiErrorID;
END_GET
SET
uiErrorID := ErrorID;
END_SET
END_PROPERTY

PROPERTY ErrorLevel : E_ErrorLevel
GET
ErrorLevel := eErrorLevel;
END_GET
SET
eErrorLevel := ErrorLevel;
END_SET
END_PROPERTY

PROPERTY ErrorMessage : STRING
GET
ErrorMessage := sErrorMessage;
END_GET
SET
sErrorMessage := ErrorMessage;
END_SET
END_PROPERTY

PROPERTY ErrorOwner : STRING
GET
ErrorOwner := sErrorOwner;
END_GET
SET
sErrorOwner := ErrorOwner;
END_SET
END_PROPERTY

//FB_Init ist immer implizit verfügbar und wird primär für die Initialisierung verwendet.
//Der Rückgabewert wird nicht ausgewertet. Für gezielte Einflussnahme können Sie
//die Methoden explizit deklarieren und darin mit dem Standard-Initialisierungscode 
//zusätzlichen Code bereitstellen. Sie können den Rückgabewert auswerten.
METHOD FB_Init: BOOL
VAR_INPUT    
	bInitRetains					: BOOL; 					// TRUE: Die Retain-Variablen werden initialisiert (Reset warm / Reset kalt)    
	bInCopyCode						: BOOL;  					// TRUE: Die Instanz wird danach in den Kopiercode kopiert (Online-Change)
	
	I_Name                : STRING;         //  Name
	I_ID                  : UINT;           // ID
//  I_itfOwner					  : ITF_Owner;      // owner 
END_VAR

Name          := I_Name;
ID            := I_ID;
END_METHOD

PROPERTY ID : UINT
GET
ID := uiID;
END_GET
SET
uiID := ID;
END_SET
END_PROPERTY

PROPERTY Init : BOOL
GET
Init := bInit;
END_GET
SET
bInit := Init;
END_SET
END_PROPERTY

METHOD mClearError : BOOL
VAR_INPUT
END_VAR

bError       		:= FALSE;
eErrorLevel  		:= E_ErrorLevel.NONE;
sErrorMessage   := '';
sErrorOwner  		:= '';

mClearError  		:= TRUE;
END_METHOD

METHOD mEnable : BOOL
VAR_INPUT
END_VAR

IF NOT bEnable THEN
    mEnable := FALSE;
    RETURN;
END_IF

IF bError THEN
    mEnable := FALSE;
    RETURN;
END_IF

mEnable := TRUE;
END_METHOD

METHOD mError : BOOL
VAR_INPUT
	I_sMessage   : STRING;
	I_eLevel		 : E_ErrorLevel;
	I_uiError		 : UINT;
END_VAR

stError.bActive				:= TRUE;
stError.eLevel				:= I_eLevel;
stError.uiErrorID			:= I_eLevel; 

stError.sOwner    		:= Name;
stError.sMessage			:= I_sMessage;

// Build full error message
stError.sFullMessage  := Concat(Name,':');
stError.sFullMessage  := Concat(stError.sFullMessage, I_sMessage);

// Error nur bei high oder critical Fehlern setzen
IF (I_eLevel = E_ErrorLevel.High)OR 
   (I_eLevel = E_ErrorLevel.Critical) 
	  	THEN
    		Error := TRUE;
END_IF

mError := TRUE;
END_METHOD

METHOD mInit : BOOL
VAR_INPUT

END_VAR

bBusy 					:= FALSE;
bDone 					:= FALSE;
bError 					:= FALSE;
sErrorMessage 	:= '';

mInit 					:= TRUE;
END_METHOD

METHOD mReset : BOOL
VAR_INPUT

END_VAR

bError 					:= FALSE;
bBusy 					:= FALSE;
bDone 					:= FALSE;
sErrorMessage 	:= '';

mReset 					:= TRUE;
END_METHOD

METHOD mVisu : BOOL
VAR_INPUT
END_VAR

mVisu:= TRUE;
END_METHOD

PROPERTY Name : string
GET
Name := sName;
END_GET
SET
sName := Name;
END_SET
END_PROPERTY

END_FUNCTION_BLOCK

// ---- 002 POUs/01 Lib/01 Device/FD_ConvoyerDevice.TcPOU
FUNCTION_BLOCK FD_ConvoyerDevice EXTENDS FD_Device IMPLEMENTS ITF_Convoyer
VAR_INPUT
END_VAR

VAR_OUTPUT
END_VAR

VAR 
	//===================== Variable
	eSource 						 : E_Convoyer;
  eDestination 				 : E_Convoyer;
	
	bRouteRequest				 : BOOL;
	bCarrierWaiting   	 : BOOL;
	bRouteGranted 			 : BOOL;
	
	bTranspOutRequest    : BOOL;
	bTranspOutBusy       : BOOL;
	bTranspOutDone       : BOOL;
	
	//===================== Instance
	fbStopperCarrieConvoyer						: FB_PneuCyl_Stopper  (GVL_Customer.C_Name_StopperCarrieConvoyer,
																													GVL_Customer.C_ID_StopperCarrieConvoyer
																										  		);																												
																												
	fbMotorConvoyer										: FB_SimpleMotor      (GVL_Customer.C_Name_ConvoyerDcMotor,
																													 GVL_Customer.C_ID_MotorComvoyer
																										  		);
																													
	fbReadHead												: FB_ReadHead        	(GVL_Customer.C_Name_ReadHead,
																													GVL_Customer.C_ID_ReadHead
																										  		); 
																													
END_VAR

VAR CONSTANT
	// --------------------------Base------------------
	C_SeqStep_OnBasePos_Start															: UINT :=  1; 
	C_SeqStep_OnBasePos_WaitOpMode												: UINT :=  2;
	C_SeqStep_OnBasePos_Done															: UINT :=  30; 
	
	// --------------------------Auto Sequence------------------
	C_SeqStep_Auto_Start																	: UINT :=  10;
	C_SeqStep_Auto_Wait_Carrier_At_Stopper								: UINT :=  110;
	C_SeqStep_Auto_Read_Destination_Once									: UINT :=  120;
	C_SeqStep_Auto_Ask_RouteManager_For_A_Route						: UINT :=  130;
	C_SeqStep_Auto_Inject_Carrier_IntoGranted_Route				: UINT :=  140;
	C_SeqStep_Auto_End																		: UINT :=  150;
	
END_VAR


//******* Important and necessary
SUPER^();  
//====================================
IF NOT Enable THEN RETURN; END_IF

fbStopperCarrieConvoyer();
fbMotorConvoyer();
fbReadHead();

PROPERTY CarrierWaiting : BOOL
GET
CarrierWaiting := bCarrierWaiting;
END_GET
SET
bCarrierWaiting := CarrierWaiting;
END_SET
END_PROPERTY

PROPERTY Destination : E_Convoyer
GET
Destination := eDestination;
END_GET
SET
eDestination := Destination;
END_SET
END_PROPERTY

//FB_Init ist immer implizit verfügbar und wird primär für die Initialisierung verwendet.
//Der Rückgabewert wird nicht ausgewertet. Für gezielte Einflussnahme können Sie
//die Methoden explizit deklarieren und darin mit dem Standard-Initialisierungscode 
//zusätzlichen Code bereitstellen. Sie können den Rückgabewert auswerten.
METHOD FB_Init: BOOL
VAR_INPUT    
	bInitRetains					: BOOL; 					// TRUE: Die Retain-Variablen werden initialisiert (Reset warm / Reset kalt)    
	bInCopyCode						: BOOL;  					// TRUE: Die Instanz wird danach in den Kopiercode kopiert (Online-Change)
	
	I_Name                : STRING;         //  Name
	I_ID                  : UINT;           // ID
  I_itfOwner					  : ITF_Owner;      // owner 
	I_eConvoyerID					: E_Convoyer;			// Source ID
END_VAR
  
	eSource := I_eConvoyerID;
END_METHOD

METHOD mAutomatic : E_CmdState
VAR_INPUT
	I_bExecute	: BOOL;
END_VAR

SUPER^.mAutomatic(TRUE);
END_METHOD

METHOD mCmdExec_Auto : E_CmdState
VAR_INPUT
END_VAR

VAR
    L_eCmd 			: E_CmdState;
END_VAR

CASE SequenceID OF

  //******************************************************* Idle 
  C_SeqStep_Idle: 
  	SequenceID       :=  C_SeqStep_Start;
  
  //****************************************************** Start
  C_SeqStep_Start:
		bRouteRequest 			:= FALSE;
    bRouteGranted 			:= FALSE;
    bTranspOutRequest 	:= FALSE;
    bTranspOutDone 			:= FALSE; 	
  	SequenceID          := C_SeqStep_Auto_Wait_Carrier_At_Stopper;
		
	C_SeqStep_Auto_Wait_Carrier_At_Stopper :
	
		IF fbStopperCarrieConvoyer.CarriePresent 
			THEN
			//eSource		 := fbReadHead.GetSource; // Get Souce if carrie present 
      	SequenceID := C_SeqStep_Auto_Read_Destination_Once;
  	END_IF
	
	C_SeqStep_Auto_Read_Destination_Once:
	// Read destination one.
  	IF fbReadHead.mRead(TRUE) = E_CmdState.Succeeded 
			THEN
  	    eDestination 		:= fbReadHead.ReadDestination;
  	    SequenceID 			:= C_SeqStep_Auto_Ask_RouteManager_For_A_Route;
  	END_IF
	
	C_SeqStep_Auto_Ask_RouteManager_For_A_Route:
	// Ask RouteManager for a route.
 		bRouteRequest := TRUE;
		
    IF bRouteGranted 
			THEN
    		bTranspOutRequest  := TRUE;
    	  SequenceID         := C_SeqStep_Auto_Inject_Carrier_IntoGranted_Route;
    	END_IF

	 C_SeqStep_Auto_Inject_Carrier_IntoGranted_Route:
      // Inject carrier into granted route.				
		IF mCmdExec_TranspOut(bTranspOutRequest ) = E_CmdState.Succeeded 
			THEN
      	bRouteRequest     := FALSE;
      	bRouteGranted     := FALSE;
      	bTranspOutRequest := FALSE;
      	SequenceID        := C_SeqStep_Auto_End;
     END_IF
									
  C_SeqStep_Error: 
    //************* all FB reset
 
 	C_SeqStep_Auto_End:
	  //**********************End 
		SequenceID := C_SeqStep_Start;
  		
END_CASE
END_METHOD

METHOD mCmdExec_BasePos : E_CmdState
VAR_INPUT
END_VAR

CASE SequenceID OF
  //******************************************************* Idle 
  C_SeqStep_Idle: 
  	;
  //****************************************************** Start
  C_SeqStep_OnBasePos_Start:
	// Home position for LTU is MIDDLE.
		fbMotorConvoyer.mStopMotor(TRUE);
		IF E_CmdState.Succeeded  = fbStopperCarrieConvoyer.mCallBase(TRUE)
			THEN
				Homed := TRUE;
  	  	Ready := TRUE;
  	  	SequenceID := C_SeqStep_OnBasePos_Done;
		END_IF
		
  C_SeqStep_Error: 
    //************* all FB reset
    mCmdExec_BasePos := mDone(); 
  //**********************Done
 	C_SeqStep_OnBasePos_Done:
  	mCmdExec_BasePos := mDone();
END_CASE
END_METHOD

METHOD mCmdExec_Service : E_CmdState
VAR_INPUT
END_VAR
;
END_METHOD

METHOD mCmdExec_TranspOut : E_CmdState
VAR_INPUT
	I_bExecute 			: BOOL;
END_VAR

IF NOT I_bExecute 
	THEN
    bTranspOutBusy := FALSE;
    mCmdExec_TranspOut := E_CmdState.Idle;
    RETURN;
END_IF

// Route not granted yet.
// Route noch nicht freigegeben
IF NOT bRouteGranted 
	THEN
  	mCmdExec_TranspOut := E_CmdState.NotReady;
    RETURN;
END_IF

bTranspOutBusy := TRUE;
bTranspOutDone := FALSE;

// Open stopper: stopper down = carrier can pass.
fbStopperCarrieConvoyer.mCallWork(TRUE);

// Start conveyor motor.
fbMotorConvoyer.mStartMotor(TRUE);

// Wait until carrier leaves stopper sensor.
IF NOT fbStopperCarrieConvoyer.CarriePresent 
	THEN
  	// Stop local injection.
  	fbMotorConvoyer.mStopMotor(TRUE);
		
  	// Close stopper again.
  	fbStopperCarrieConvoyer.mCallBase(TRUE);
  	bTranspOutBusy := FALSE;
  	bTranspOutDone := TRUE;
  	mCmdExec_TranspOut := E_CmdState.Succeeded;
  	RETURN;
END_IF
END_METHOD

METHOD mHold : E_CmdState
VAR_INPUT
	I_bExecute	: BOOL;
END_VAR
END_METHOD

METHOD mHome : E_CmdState
VAR_INPUT
	I_bExecute	: BOOL;
END_VAR
SUPER^.mHome(I_bExecute);
END_METHOD

METHOD mRelease : E_CmdState
VAR_INPUT
	I_bExecute	: BOOL;
END_VAR
END_METHOD

METHOD mSequence : E_CmdState
VAR_INPUT
	I_bExecute				: BOOL;
END_VAR

VAR
	L_eState 					: E_CmdState;
END_VAR
mSequence := SUPER^.mSequence(I_bExecute);	


// Generic checks from parent
L_eState := SUPER^.mSequence(I_bExecute := I_bExecute);

IF L_eState <> E_CmdState.Busy 
	THEN
    mSequence := L_eState;
    RETURN;
END_IF

CASE Mode OF
	E_Mode.Homing:
		mSequence := mCmdExec_BasePos();
	E_Mode.Auto:
		mSequence := mCmdExec_Auto();
	E_Mode.Service:
		mSequence := mCmdExec_Service();	
END_CASE
END_METHOD

METHOD mService : E_CmdState
VAR_INPUT
	I_bExecute	: BOOL;
END_VAR
END_METHOD

METHOD mStop : E_CmdState
VAR_INPUT
	I_bExecute	: BOOL;
END_VAR
END_METHOD

PROPERTY RouteGranted : BOOL
GET
RouteGranted := bRouteGranted;
END_GET
SET
bRouteGranted := RouteGranted;
END_SET
END_PROPERTY

PROPERTY RouteRequest : BOOL
GET
RouteRequest := bRouteRequest;
END_GET
SET
bRouteRequest := RouteRequest;
END_SET
END_PROPERTY

PROPERTY Source : E_Convoyer
GET
Source := eSource;
END_GET
SET
eSource := Source;
END_SET
END_PROPERTY

PROPERTY TranspOutBusy : BOOL
GET
TranspOutBusy := bTranspOutBusy;
END_GET
SET
bTranspOutBusy := TranspOutBusy;
END_SET
END_PROPERTY

PROPERTY TranspOutDone : BOOL
GET
TranspOutDone := bTranspOutDone;
END_GET
SET
bTranspOutDone := TranspOutDone;
END_SET
END_PROPERTY

PROPERTY TranspOutRequest : BOOL
GET
TranspOutRequest := bTranspOutRequest;
END_GET
SET
bTranspOutRequest := TranspOutRequest;
END_SET
END_PROPERTY

END_FUNCTION_BLOCK

// ---- 002 POUs/01 Lib/02 SimpleDevice/FB_PneuCyl_Stopper.TcPOU
FUNCTION_BLOCK FB_PneuCyl_Stopper EXTENDS FB_Base
VAR_INPUT
		bCarriePresent1										: BOOL;
END_VAR
VAR_OUTPUT
END_VAR
VAR
	//================================= Variable
	bCarriePresent										: BOOL;
	bHmiSimCarrie 										: BOOL;

	
	//================================= Instance
	fbStopperOut											: FB_Output					(GVL_Customer.C_Name_StopperOut,
																												 GVL_Customer.C_ID_StopperOut
																											  );
	
	fbStopperOccupied									: FB_Input					(GVL_Customer.C_Name_StopperOccupied,
																												 GVL_Customer.C_ID_StopperOccupied
																											  );
END_VAR

//================== Must!!
SUPER^();  
IF NOT Enable THEN RETURN; END_IF;
// Check Carrie available
bCarriePresent := fbStopperOccupied.bBoolValue OR bHmiSimCarrie ;

PROPERTY CarriePresent : BOOL
GET
CarriePresent := bCarriePresent;
END_GET
SET
bCarriePresent := CarriePresent;
END_SET
END_PROPERTY

//FB_Init ist immer implizit verfügbar und wird primär für die Initialisierung verwendet.
//Der Rückgabewert wird nicht ausgewertet. Für gezielte Einflussnahme können Sie
//die Methoden explizit deklarieren und darin mit dem Standard-Initialisierungscode 
//zusätzlichen Code bereitstellen. Sie können den Rückgabewert auswerten.
METHOD FB_Init: BOOL
VAR_INPUT    
	bInitRetains					: BOOL; 					// TRUE: Die Retain-Variablen werden initialisiert (Reset warm / Reset kalt)    
	bInCopyCode						: BOOL;  					// TRUE: Die Instanz wird danach in den Kopiercode kopiert (Online-Change)
	
	I_Name                : STRING;         //  Name
	I_ID                  : UINT;            // ID
END_VAR
END_METHOD

METHOD mCallBase : E_CmdState
VAR_INPUT
	I_bExecute			 : BOOL;
END_VAR
// No command requested.
IF NOT I_bExecute 
	THEN
    mCallBase  := E_CmdState.Idle;
    RETURN;
END_IF

// Base position:
// stopper up = carrier is blocked.
fbStopperOut.bBoolValue := FALSE;
mCallBase := E_CmdState.Succeeded;
END_METHOD

METHOD mCallWork : E_CmdState
VAR_INPUT
	I_bExecute			 : BOOL;
END_VAR
// No command requested.
IF NOT I_bExecute 
	THEN
    mCallWork  := E_CmdState.Idle;
    RETURN;
END_IF

// Base position:
// stopper Down = carrier is free.
fbStopperOut.bBoolValue := TRUE;
mCallWork := E_CmdState.Succeeded;
END_METHOD

END_FUNCTION_BLOCK

// ---- 002 POUs/01 Lib/Digit I_O/Output/FB_Output.TcPOU
FUNCTION_BLOCK FB_Output EXTENDS FB_Base
VAR_INPUT
	bBoolValue								: BOOL;
END_VAR
VAR_OUTPUT
	
END_VAR
VAR
	bQAT_HardwareLink	AT %Q*	:	BOOL; // hardware link
	
END_VAR


SUPER^();

bQAT_HardwareLink := bBoolValue;

//FB_Init ist immer implizit verfügbar und wird primär für die Initialisierung verwendet.
//Der Rückgabewert wird nicht ausgewertet. Für gezielte Einflussnahme können Sie
//die Methoden explizit deklarieren und darin mit dem Standard-Initialisierungscode 
//zusätzlichen Code bereitstellen. Sie können den Rückgabewert auswerten.
METHOD FB_Init: BOOL
VAR_INPUT    
	bInitRetains					: BOOL; 					// TRUE: Die Retain-Variablen werden initialisiert (Reset warm / Reset kalt)    
	bInCopyCode						: BOOL;  					// TRUE: Die Instanz wird danach in den Kopiercode kopiert (Online-Change)
	
	I_Name                : STRING;         //  Name
	I_ID                  : UINT;            // ID
END_VAR
END_METHOD

END_FUNCTION_BLOCK

// ---- 002 POUs/01 Lib/02 SimpleDevice/FB_ReadHead.TcPOU
FUNCTION_BLOCK FB_ReadHead EXTENDS FB_Base
VAR_INPUT
END_VAR
VAR_OUTPUT
END_VAR
VAR
	//eGetSource									: E_Convoyer;
	eReadDestination						: E_Convoyer;
	bExecute										: BOOL;
	fbDrand											: DRAND;
	aDestinationListe      			: ARRAY[1..4] OF UINT := [3, 6, 9, 12];
	
END_VAR

//================== Must!!
SUPER^();  
IF NOT Enable THEN RETURN; END_IF;

PROPERTY Execute : BOOL
GET
Execute := bExecute;
END_GET
SET
bExecute := Execute;
END_SET
END_PROPERTY

//FB_Init ist immer implizit verfügbar und wird primär für die Initialisierung verwendet.
//Der Rückgabewert wird nicht ausgewertet. Für gezielte Einflussnahme können Sie
//die Methoden explizit deklarieren und darin mit dem Standard-Initialisierungscode 
//zusätzlichen Code bereitstellen. Sie können den Rückgabewert auswerten.
METHOD FB_Init: BOOL
VAR_INPUT    
	bInitRetains					: BOOL; 					// TRUE: Die Retain-Variablen werden initialisiert (Reset warm / Reset kalt)    
	bInCopyCode						: BOOL;  					// TRUE: Die Instanz wird danach in den Kopiercode kopiert (Online-Change)
	
	I_Name                : STRING;         //  Name
	I_ID                  : UINT;            // ID
END_VAR
END_METHOD

METHOD mRead : E_CmdState
VAR_INPUT
	I_bExecute		: BOOL;
END_VAR

VAR
	L_uiReadData					: UINT;
	L_uiIndex							: INT;
	
END_VAR

IF NOT I_bExecute 
	THEN
    mRead := E_CmdState.Idle;
    RETURN;
END_IF

fbDrand(); 
L_uiIndex			:= LREAL_TO_INT(((fbDrand.Num) * 4)+1);
IF L_uiIndex < 1 THEN L_uiIndex := 1; END_IF;
IF L_uiIndex > 4 THEN L_uiIndex := 4; END_IF;
L_uiReadData 	:= aDestinationListe[L_uiIndex];
bExecute			:= FALSE;

CASE L_uiReadData OF
	3 : eReadDestination  := E_Convoyer.Convoyer_3;
	6 : eReadDestination 	:= E_Convoyer.Convoyer_6; 
	9 : eReadDestination 	:= E_Convoyer.Convoyer_9;
 12 : eReadDestination 	:= E_Convoyer.Convoyer_12;
ELSE
    mRead 						:= E_CmdState.Error;
    RETURN;
END_CASE

mRead := E_CmdState.Succeeded;
END_METHOD

PROPERTY ReadDestination : E_Convoyer
GET
ReadDestination := eReadDestination;
END_GET
SET
eReadDestination := ReadDestination;
END_SET
END_PROPERTY

END_FUNCTION_BLOCK

// ---- 002 POUs/01 Lib/01 Device/FD_RouteManagerDevice.TcPOU
(*
 receive a request : source on destination
 calculate the  path
 verify required resources
 reserve the relevant Ltu or conveyors
 give a ST_Route to the route executor
*)

FUNCTION_BLOCK FD_RouteManagerDevice EXTENDS FD_Device IMPLEMENTS ITF_RouteProvider
VAR_INPUT
END_VAR

VAR_OUTPUT
END_VAR

VAR
	//===================== interface
 	itfLTU3  											: ITF_LTU;
 	itfLTU6  											: ITF_LTU;
 	itfLTU9  											: ITF_LTU;
 	itfLTU12 											: ITF_LTU;
          											
	itfC3    											: ITF_Convoyer;
	itfC6    											: ITF_Convoyer;
	itfC9    											: ITF_Convoyer;
	itfC12   											: ITF_Convoyer;
	
	//===================== Variable
  //eSource			 									: E_Convoyer;
  //eDestination 									: E_Convoyer;
	
	astRouteQueue 								: ARRAY[1..10] OF ST_RouteJob; // Warteschlange speichern die berechneteten route 
	uiNextJobID 									: UINT := 1;
	
//	bRouteRequest   							: BOOL;
//	bRouteAvailable 							: BOOL;
//  bRouteReserved								: BOOL;
	
	//===================== Instance
																								
END_VAR

VAR CONSTANT
		// --------------------------Base------------------
	C_SeqStep_OnBasePos_Start								: UINT :=  1; 
	C_SeqStep_OnBasePos_Error								: UINT :=  30;
	C_SeqStep_OnBasePos_Done								: UINT :=  100; 
	
	// --------------------------Auto Sequence------------------
	
	C_SeqStep_Auto_Start										: UINT :=  1;
	C_SeqStep_Auto_End											: UINT :=  2;
END_VAR


//******* Important and necessary
SUPER^();  
//====================================
IF NOT Enable THEN RETURN; END_IF

//FB_Init ist immer implizit verfügbar und wird primär für die Initialisierung verwendet.
//Der Rückgabewert wird nicht ausgewertet. Für gezielte Einflussnahme können Sie
//die Methoden explizit deklarieren und darin mit dem Standard-Initialisierungscode 
//zusätzlichen Code bereitstellen. Sie können den Rückgabewert auswerten.
METHOD FB_Init: BOOL
VAR_INPUT    
	bInitRetains					: BOOL; 					// TRUE: Die Retain-Variablen werden initialisiert (Reset warm / Reset kalt)    
	bInCopyCode						: BOOL;  					// TRUE: Die Instanz wird danach in den Kopiercode kopiert (Online-Change)
	
	I_Name                : STRING;         //  Name
	I_ID                  : UINT;           // ID
  I_itfOwner					  : ITF_Owner;      // owner 
	
// ITF_LTU	
	I_itfLTU3  						: ITF_LTU;        
 	I_itfLTU6  						: ITF_LTU;
 	I_itfLTU9  						: ITF_LTU;
 	I_itfLTU12 						: ITF_LTU;
  
// ITF_Convoyer  							
	I_itfC3    						: ITF_Convoyer;
	I_itfC6    						: ITF_Convoyer;
	I_itfC9    						: ITF_Convoyer;
	I_itfC12   						: ITF_Convoyer;
END_VAR

// chek and link LTU
IF I_itfLTU3  <>0 THEN itfLTU3  := I_itfLTU3; END_IF
IF I_itfLTU6  <>0 THEN itfLTU6  := I_itfLTU6; END_IF
IF I_itfLTU9  <>0 THEN itfLTU9  := I_itfLTU9; END_IF
IF I_itfLTU12 <>0 THEN itfLTU12 := I_itfLTU12;END_IF

// chek and link covoyer
IF I_itfC3  <>0 THEN itfC3  := I_itfC3; END_IF
IF I_itfC6  <>0 THEN itfC6  := I_itfC6; END_IF
IF I_itfC9  <>0 THEN itfC9  := I_itfC9; END_IF
IF I_itfC12 <>0 THEN itfC12 := I_itfC12;END_IF
END_METHOD

METHOD mAutomatic : E_CmdState
VAR_INPUT
	I_bExecute	: BOOL;
END_VAR

SUPER^.mAutomatic(TRUE);
END_METHOD

METHOD PROTECTED mBuildRoute : BOOL
VAR_INPUT
	I_eSource       : E_Convoyer;
	I_eDestination  : E_Convoyer;
	I_refstRoute    : REFERENCE TO ST_Route;
END_VAR

// Reset route.
I_refstRoute.eSource      := I_eSource;
I_refstRoute.eDestination := I_eDestination;
I_refstRoute.iuStepCount  := 0;

//==================================================
// R3 -> 3
// C3 -> LTU3 -> LTU6
//==================================================
IF (I_eSource = E_Convoyer.Convoyer_3)
	AND (I_eDestination = E_Convoyer.Convoyer_3) 
		THEN
    	I_refstRoute.iuStepCount := 2;
			
    	I_refstRoute.astSteps[1].eConvoyer    := E_Convoyer.Convoyer_3;
    	I_refstRoute.astSteps[1].eLTUPosition := E_LTUPosition.LTU_TOP;
    	
    	I_refstRoute.astSteps[2].eConvoyer    := E_Convoyer.Convoyer_6;
    	I_refstRoute.astSteps[2].eLTUPosition := E_LTUPosition.LTU_TOP;
    	
    	mBuildRoute := TRUE;
    	RETURN;
END_IF

//==================================================
// R3 -> 6
// C3 -> LTU3 -> LTU6 -> bottom -> C6
//==================================================
IF (I_eSource = E_Convoyer.Convoyer_3)
   AND (I_eDestination = E_Convoyer.Convoyer_6) 
	 	THEN
    	I_refstRoute.iuStepCount := 3;
    	
    	I_refstRoute.astSteps[1].eConvoyer     := E_Convoyer.Convoyer_3;
    	I_refstRoute.astSteps[1].eLTUPosition  := E_LTUPosition.LTU_TOP;
    	
    	I_refstRoute.astSteps[2].eConvoyer     := E_Convoyer.Convoyer_6;
    	I_refstRoute.astSteps[2].eLTUPosition  := E_LTUPosition.LTU_TOP;
    	
    	I_refstRoute.astSteps[3].eConvoyer     := E_Convoyer.Convoyer_6;
    	I_refstRoute.astSteps[3].eLTUPosition  := E_LTUPosition.LTU_BOTTOM;
    	
    	mBuildRoute := TRUE;
    RETURN;
END_IF

// R3 -> 9
// C3 -> LTU6 bottom -> LTU9 top -> LTU12 -> C9
//==================================================
IF (I_eSource = E_Convoyer.Convoyer_3)
   AND (I_eDestination = E_Convoyer.Convoyer_9) 
	 	THEN
    	I_refstRoute.iuStepCount := 6;
    	
    	I_refstRoute.astSteps[1].eConvoyer     := E_Convoyer.Convoyer_3;
    	I_refstRoute.astSteps[1].eLTUPosition  := E_LTUPosition.LTU_TOP;
    	
    	I_refstRoute.astSteps[2].eConvoyer     := E_Convoyer.Convoyer_6;
    	I_refstRoute.astSteps[2].eLTUPosition  := E_LTUPosition.LTU_TOP;
    	
    	I_refstRoute.astSteps[3].eConvoyer     := E_Convoyer.Convoyer_6;
    	I_refstRoute.astSteps[3].eLTUPosition  := E_LTUPosition.LTU_BOTTOM;
    	
    	I_refstRoute.astSteps[4].eConvoyer     := E_Convoyer.Convoyer_9;
    	I_refstRoute.astSteps[4].eLTUPosition  := E_LTUPosition.LTU_BOTTOM;
    	
    	I_refstRoute.astSteps[5].eConvoyer     := E_Convoyer.Convoyer_9;
    	I_refstRoute.astSteps[5].eLTUPosition  := E_LTUPosition.LTU_TOP;
    	
    	I_refstRoute.astSteps[6].eConvoyer     := E_Convoyer.Convoyer_12;
    	I_refstRoute.astSteps[6].eLTUPosition  := E_LTUPosition.LTU_TOP;
    	
    	mBuildRoute := TRUE;
			RETURN;
END_IF

//==================================================
// R3 -> 12
// C3 -> LTU3 -> bottom -> C12
// Needs LTU3 only
//==================================================
IF (I_eSource = E_Convoyer.Convoyer_3)
   AND (I_eDestination = E_Convoyer.Convoyer_12) 
	 THEN
   	I_refstRoute.iuStepCount := 1;
		
   	I_refstRoute.astSteps[1].eConvoyer 		:= E_Convoyer.Convoyer_3;
   	I_refstRoute.astSteps[1].eLTUPosition  := E_LTUPosition.LTU_BOTTOM;
   	
   	mBuildRoute := TRUE;
   	RETURN;
END_IF

//==================================================
// R6 -> 6
// C6 line, BOTTOM continuity LTU6 + LTU9
//==================================================
IF (I_eSource = E_Convoyer.Convoyer_6)
   AND (I_eDestination = E_Convoyer.Convoyer_6) 
   	THEN
    I_refstRoute.iuStepCount := 2;

    I_refstRoute.astSteps[1].eConvoyer     := E_Convoyer.Convoyer_6;
    I_refstRoute.astSteps[1].eLTUPosition  := E_LTUPosition.LTU_BOTTOM;

    I_refstRoute.astSteps[2].eConvoyer     := E_Convoyer.Convoyer_9;
    I_refstRoute.astSteps[2].eLTUPosition  := E_LTUPosition.LTU_BOTTOM;

    mBuildRoute := TRUE;
    RETURN;
END_IF

//==================================================
// R6 -> 3
// C6 -> LTU6 -> top -> C3
// Needs LTU6 only
//==================================================
IF (I_eSource = E_Convoyer.Convoyer_6)
   AND (I_eDestination = E_Convoyer.Convoyer_3) 
   	THEN
    I_refstRoute.iuStepCount := 1;

    I_refstRoute.astSteps[1].eConvoyer     := E_Convoyer.Convoyer_6;
    I_refstRoute.astSteps[1].eLTUPosition  := E_LTUPosition.LTU_TOP;

    mBuildRoute := TRUE;
    RETURN;
END_IF

//==================================================
// R6 -> 9
// C6 -> LTU6 -> LTU9 -> top -> LTU12 -> C9
//==================================================
IF (I_eSource = E_Convoyer.Convoyer_6)
   AND (I_eDestination = E_Convoyer.Convoyer_9) 
   	THEN
    	I_refstRoute.iuStepCount := 4;
    	
    	I_refstRoute.astSteps[1].eConvoyer     := E_Convoyer.Convoyer_6;
    	I_refstRoute.astSteps[1].eLTUPosition  := E_LTUPosition.LTU_BOTTOM;
    	
    	I_refstRoute.astSteps[2].eConvoyer     := E_Convoyer.Convoyer_9;
    	I_refstRoute.astSteps[2].eLTUPosition  := E_LTUPosition.LTU_BOTTOM;
    	
    	I_refstRoute.astSteps[3].eConvoyer     := E_Convoyer.Convoyer_9;
    	I_refstRoute.astSteps[3].eLTUPosition  := E_LTUPosition.LTU_TOP;
    	
    	I_refstRoute.astSteps[4].eConvoyer     := E_Convoyer.Convoyer_12;
    	I_refstRoute.astSteps[4].eLTUPosition  := E_LTUPosition.LTU_TOP;
    	
    	mBuildRoute := TRUE;
    	RETURN;
END_IF

//==================================================
// R6 -> 12
// C6 -> LTU9 top -> LTU12 bottom -> C12
//==================================================
IF (I_eSource = E_Convoyer.Convoyer_6)
   AND (I_eDestination = E_Convoyer.Convoyer_12) 
   	THEN
    	I_refstRoute.iuStepCount := 6;
    	
    	I_refstRoute.astSteps[1].eConvoyer     := E_Convoyer.Convoyer_6;
    	I_refstRoute.astSteps[1].eLTUPosition  := E_LTUPosition.LTU_BOTTOM;
    	
    	I_refstRoute.astSteps[2].eConvoyer     := E_Convoyer.Convoyer_9;
    	I_refstRoute.astSteps[2].eLTUPosition  := E_LTUPosition.LTU_BOTTOM;
    	
    	I_refstRoute.astSteps[3].eConvoyer     := E_Convoyer.Convoyer_9;
    	I_refstRoute.astSteps[3].eLTUPosition  := E_LTUPosition.LTU_TOP;
    	
    	I_refstRoute.astSteps[4].eConvoyer     := E_Convoyer.Convoyer_12;
    	I_refstRoute.astSteps[4].eLTUPosition  := E_LTUPosition.LTU_TOP;
    	
    	I_refstRoute.astSteps[5].eConvoyer     := E_Convoyer.Convoyer_12;
    	I_refstRoute.astSteps[5].eLTUPosition  := E_LTUPosition.LTU_BOTTOM;
    	
    	I_refstRoute.astSteps[6].eConvoyer     := E_Convoyer.Convoyer_3;
    	I_refstRoute.astSteps[6].eLTUPosition  := E_LTUPosition.LTU_BOTTOM;
    	
    	mBuildRoute := TRUE;
    	RETURN;
END_IF

//==================================================
// R9 -> 9
// C9 line, TOP continuity LTU9 + LTU12
//==================================================
IF (I_eSource = E_Convoyer.Convoyer_9)
   AND (I_eDestination = E_Convoyer.Convoyer_9) 
   	THEN
    	I_refstRoute.iuStepCount := 2;
    	
    	I_refstRoute.astSteps[1].eConvoyer     := E_Convoyer.Convoyer_9;
    	I_refstRoute.astSteps[1].eLTUPosition  := E_LTUPosition.LTU_TOP;
    	
    	I_refstRoute.astSteps[2].eConvoyer     := E_Convoyer.Convoyer_12;
    	I_refstRoute.astSteps[2].eLTUPosition  := E_LTUPosition.LTU_TOP;
    	
    	mBuildRoute := TRUE;
    	RETURN;
END_IF

//==================================================
// R9 -> 3
// C9 -> LTU12 bottom -> LTU3 top -> LTU6 -> C3
//==================================================
IF (I_eSource = E_Convoyer.Convoyer_9)
   AND (I_eDestination = E_Convoyer.Convoyer_3) 
   	THEN
    	I_refstRoute.iuStepCount := 6;
    	
    	I_refstRoute.astSteps[1].eConvoyer     := E_Convoyer.Convoyer_9;
    	I_refstRoute.astSteps[1].eLTUPosition  := E_LTUPosition.LTU_TOP;
    	
    	I_refstRoute.astSteps[2].eConvoyer     := E_Convoyer.Convoyer_12;
    	I_refstRoute.astSteps[2].eLTUPosition  := E_LTUPosition.LTU_TOP;
    	
    	I_refstRoute.astSteps[3].eConvoyer     := E_Convoyer.Convoyer_12;
    	I_refstRoute.astSteps[3].eLTUPosition  := E_LTUPosition.LTU_BOTTOM;
    	
    	I_refstRoute.astSteps[4].eConvoyer     := E_Convoyer.Convoyer_3;
    	I_refstRoute.astSteps[4].eLTUPosition  := E_LTUPosition.LTU_BOTTOM;
    	
    	I_refstRoute.astSteps[5].eConvoyer     := E_Convoyer.Convoyer_3;
    	I_refstRoute.astSteps[5].eLTUPosition  := E_LTUPosition.LTU_TOP;
    	
    	I_refstRoute.astSteps[6].eConvoyer     := E_Convoyer.Convoyer_6;
    	I_refstRoute.astSteps[6].eLTUPosition  := E_LTUPosition.LTU_TOP;

    	mBuildRoute := TRUE;
   	  RETURN;
END_IF

//==================================================
// R9 -> 6
// C9 -> LTU9 -> bottom -> C6
// Needs LTU9 only
//==================================================
IF (I_eSource = E_Convoyer.Convoyer_9)
   AND (I_eDestination = E_Convoyer.Convoyer_6) 
	 	THEN
    	I_refstRoute.iuStepCount := 1;
    	
    	I_refstRoute.astSteps[1].eConvoyer     := E_Convoyer.Convoyer_9;
    	I_refstRoute.astSteps[1].eLTUPosition  := E_LTUPosition.LTU_BOTTOM;
    	
    	mBuildRoute := TRUE;
    	RETURN;
END_IF

//==================================================
// R9 -> 12
// C9 -> LTU12 -> bottom -> C12
// Needs LTU12 + LTU3 bottom for complete C12 line
//==================================================
IF (I_eSource = E_Convoyer.Convoyer_9)
   AND (I_eDestination = E_Convoyer.Convoyer_12) 
	 	THEN
    	I_refstRoute.iuStepCount := 4;
    	
    	I_refstRoute.astSteps[1].eConvoyer     := E_Convoyer.Convoyer_9;
    	I_refstRoute.astSteps[1].eLTUPosition  := E_LTUPosition.LTU_TOP;
    	
    	I_refstRoute.astSteps[2].eConvoyer     := E_Convoyer.Convoyer_12;
    	I_refstRoute.astSteps[2].eLTUPosition  := E_LTUPosition.LTU_TOP;
    	
    	I_refstRoute.astSteps[3].eConvoyer     := E_Convoyer.Convoyer_12;
    	I_refstRoute.astSteps[3].eLTUPosition  := E_LTUPosition.LTU_BOTTOM;
    	
    	I_refstRoute.astSteps[4].eConvoyer     := E_Convoyer.Convoyer_3;
    	I_refstRoute.astSteps[4].eLTUPosition  := E_LTUPosition.LTU_BOTTOM;
    	
    	mBuildRoute := TRUE;
    	RETURN;
END_IF

//==================================================
// R12 -> 12
// C12 line, BOTTOM continuity LTU12 + LTU3
//==================================================
IF (I_eSource = E_Convoyer.Convoyer_12)
   AND (I_eDestination = E_Convoyer.Convoyer_12) 
   	THEN
    	I_refstRoute.iuStepCount := 2;
    	
    	I_refstRoute.astSteps[1].eConvoyer     := E_Convoyer.Convoyer_12;
    	I_refstRoute.astSteps[1].eLTUPosition  := E_LTUPosition.LTU_BOTTOM;
    	
    	I_refstRoute.astSteps[2].eConvoyer     := E_Convoyer.Convoyer_3;
    	I_refstRoute.astSteps[2].eLTUPosition  := E_LTUPosition.LTU_BOTTOM;
    	
    	mBuildRoute := TRUE;
    	RETURN;
END_IF

//==================================================
// R12 -> 3
// C12 -> LTU3 top -> LTU6 -> C3
//==================================================
IF (I_eSource = E_Convoyer.Convoyer_12)
   AND (I_eDestination = E_Convoyer.Convoyer_3) 
   	THEN
    	I_refstRoute.iuStepCount := 4;
    	
    	I_refstRoute.astSteps[1].eConvoyer     := E_Convoyer.Convoyer_12;
    	I_refstRoute.astSteps[1].eLTUPosition  := E_LTUPosition.LTU_BOTTOM;
    	
    	I_refstRoute.astSteps[2].eConvoyer     := E_Convoyer.Convoyer_3;
    	I_refstRoute.astSteps[2].eLTUPosition  := E_LTUPosition.LTU_BOTTOM;
    	
    	I_refstRoute.astSteps[3].eConvoyer     := E_Convoyer.Convoyer_3;
    	I_refstRoute.astSteps[3].eLTUPosition  := E_LTUPosition.LTU_TOP;
    	
    	I_refstRoute.astSteps[4].eConvoyer     := E_Convoyer.Convoyer_6;
    	I_refstRoute.astSteps[4].eLTUPosition  := E_LTUPosition.LTU_TOP;
    	
    	mBuildRoute := TRUE;
    	RETURN;
END_IF

//==================================================
// R12 -> 6
// C12 -> LTU3 top -> LTU6 bottom -> LTU9 -> C6
//==================================================
IF (I_eSource = E_Convoyer.Convoyer_12)
   AND (I_eDestination = E_Convoyer.Convoyer_6) 
   	THEN
    	I_refstRoute.iuStepCount := 6;
    	
    	I_refstRoute.astSteps[1].eConvoyer     := E_Convoyer.Convoyer_12;
    	I_refstRoute.astSteps[1].eLTUPosition  := E_LTUPosition.LTU_BOTTOM;
    	
    	I_refstRoute.astSteps[2].eConvoyer     := E_Convoyer.Convoyer_3;
    	I_refstRoute.astSteps[2].eLTUPosition  := E_LTUPosition.LTU_BOTTOM;
    	
    	I_refstRoute.astSteps[3].eConvoyer     := E_Convoyer.Convoyer_3;
    	I_refstRoute.astSteps[3].eLTUPosition  := E_LTUPosition.LTU_TOP;
    	
    	I_refstRoute.astSteps[4].eConvoyer     := E_Convoyer.Convoyer_6;
    	I_refstRoute.astSteps[4].eLTUPosition  := E_LTUPosition.LTU_TOP;
    	
    	I_refstRoute.astSteps[5].eConvoyer     := E_Convoyer.Convoyer_6;
    	I_refstRoute.astSteps[5].eLTUPosition  := E_LTUPosition.LTU_BOTTOM;
    	
    	I_refstRoute.astSteps[6].eConvoyer     := E_Convoyer.Convoyer_9;
    	I_refstRoute.astSteps[6].eLTUPosition  := E_LTUPosition.LTU_BOTTOM;
    	
    	mBuildRoute := TRUE;
    	RETURN;
END_IF

//==================================================
// R12 -> 9
// C12 -> LTU12 -> top -> C9
// Needs LTU12 only
//==================================================
IF (I_eSource = E_Convoyer.Convoyer_12)
   AND (I_eDestination = E_Convoyer.Convoyer_9) 
   	THEN
    	I_refstRoute.iuStepCount := 1;
    	
    	I_refstRoute.astSteps[1].eConvoyer     := E_Convoyer.Convoyer_12;
    	I_refstRoute.astSteps[1].eLTUPosition  := E_LTUPosition.LTU_TOP;
    	
    	mBuildRoute := TRUE;
    	RETURN;
END_IF

//==================================================
// No route found
//==================================================
mBuildRoute := FALSE;
END_METHOD

METHOD mCheckRouteFree : BOOL
VAR_INPUT
    Ref_stRoute : REFERENCE TO ST_Route;
END_VAR
VAR
	L_uiIndex : UINT;
END_VAR

mCheckRouteFree := TRUE;

//========================Check each LTU used by the route
FOR L_uiIndex := 1 TO Ref_stRoute.iuStepCount DO
	
	CASE Ref_stRoute.astSteps[L_uiIndex].eConvoyer OF
		E_Convoyer.Convoyer_3:
			IF itfLTU3.ReservedBy <> E_Convoyer.Convoyer_NONE 
				THEN
					mCheckRouteFree := FALSE;
					RETURN;
			END_IF
		E_Convoyer.Convoyer_6:
			IF itfLTU6.ReservedBy <> E_Convoyer.Convoyer_NONE  
				THEN
			    mCheckRouteFree := FALSE;
			    RETURN;
			END_IF
		E_Convoyer.Convoyer_9:
			IF itfLTU9.ReservedBy <> E_Convoyer.Convoyer_NONE 
				THEN
			    mCheckRouteFree := FALSE;
			    RETURN;
			END_IF
		E_Convoyer.Convoyer_12:
			IF itfLTU12.ReservedBy <> E_Convoyer.Convoyer_NONE 
				THEN
			  	mCheckRouteFree := FALSE;
			    RETURN;
			END_IF
	END_CASE
END_FOR
END_METHOD

METHOD mCmdExec_Auto : E_CmdState
VAR_INPUT
END_VAR
// hat kein automatique sequence
CASE SequenceID OF

  //******************************************************* Idle 
  C_SeqStep_Idle: 
  	SequenceID       :=  C_SeqStep_Auto_Start;
  
  //****************************************************** Start
  C_SeqStep_Auto_Start:
		//========================
		// Check status C3
		IF itfC3.RouteRequest AND NOT itfC3.RouteGranted
			THEN
			  IF mRequestRoute(TRUE, itfC3.Source, itfC3.Destination) = E_CmdState.Succeeded
					THEN
						itfC3.RouteGranted := TRUE;
				END_IF
		END_IF
		
		//========================
		// Check status C6
		IF itfC6.RouteRequest AND NOT itfC6.RouteGranted
			THEN
			  IF mRequestRoute(TRUE, itfC6.Source, itfC6.Destination) = E_CmdState.Succeeded
					THEN
						itfC6.RouteGranted := TRUE;
				END_IF
		END_IF
		
		//========================
		// Check status C9
		IF itfC9.RouteRequest AND NOT itfC9.RouteGranted
			THEN
			  IF mRequestRoute(TRUE, itfC9.Source, itfC9.Destination) = E_CmdState.Succeeded
					THEN
						itfC9.RouteGranted := TRUE;
				END_IF
		END_IF
		
		//========================
		// Check status C12
		IF itfC12.RouteRequest AND NOT itfC12.RouteGranted
			THEN
			  IF mRequestRoute(TRUE, itfC12.Source, itfC12.Destination) = E_CmdState.Succeeded
					THEN
						itfC12.RouteGranted := TRUE;
				END_IF
		END_IF
	
	//****************************************************** Error
  C_SeqStep_Error: 
    //************* all FB reset
		;
	//****************************************************** Error
 	C_SeqStep_Auto_End:
  	SequenceID 			 := C_SeqStep_Auto_Start;

END_CASE
END_METHOD

METHOD mCmdExec_BasePos : E_CmdState
VAR_INPUT
END_VAR

CASE SequenceID OF

  //******************************************************* Idle 
  C_SeqStep_Idle: 
  	SequenceID       := C_SeqStep_OnBasePos_Start;
  
  //****************************************************** Start
  C_SeqStep_OnBasePos_Start:
		SequenceID       := C_SeqStep_OnBasePos_Done;
	
	//****************************************************** Error
  C_SeqStep_OnBasePos_Error: 
    //************* all FB reset
    mCmdExec_BasePos := mDone(); 
		
  //****************************************************** End
 	C_SeqStep_OnBasePos_Done:
  	mCmdExec_BasePos := mDone();

END_CASE
END_METHOD

METHOD mCmdExec_Service : E_CmdState
VAR_INPUT
END_VAR

 Ready 								:= TRUE;
 SequenceBusy 				:= FALSE;
 SequenceDone 				:= TRUE;
 SequenceID 					:= C_SeqStep_Idle;
 mCmdExec_Service 		:= E_CmdState.Succeeded;
 RETURN;
END_METHOD

METHOD mGetNextRoute : E_CmdState
VAR_OUTPUT
	O_pRouteJob				: POINTER TO ST_RouteJob;
END_VAR

VAR
	L_uiIndex  : UINT;
END_VAR

// Search if first valid route job not already executing
FOR L_uiIndex := 1 TO 10 DO
	IF astRouteQueue[L_uiIndex].bValid
		 AND astRouteQueue[L_uiIndex].bReserved
		 AND NOT astRouteQueue[L_uiIndex].bExecuting
		 AND NOT astRouteQueue[L_uiIndex].bDone
		 AND NOT astRouteQueue[L_uiIndex].bError 
		 	THEN
        astRouteQueue[L_uiIndex].bExecuting := TRUE;
        O_pRouteJob   := ADR(astRouteQueue[L_uiIndex]);
        mGetNextRoute   := E_CmdState.Succeeded;
        RETURN;
   END_IF
END_FOR
mGetNextRoute := E_CmdState.Idle;
END_METHOD

METHOD mHold : E_CmdState
VAR_INPUT
	I_bExecute	: BOOL;
END_VAR

SUPER^.mHold(I_bExecute);
END_METHOD

METHOD mHome : E_CmdState
VAR_INPUT
	I_bExecute	: BOOL;
END_VAR

SUPER^.mHome(I_bExecute);
END_METHOD

METHOD mRelease : E_CmdState
VAR_INPUT
	I_bExecute	: BOOL;
END_VAR

SUPER^.mRelease(I_bExecute);
END_METHOD

METHOD mReleaseResources : BOOL
VAR_INPUT
    Ref_stRoute : REFERENCE TO ST_Route;
END_VAR
VAR
	L_uiIndex : UINT;
END_VAR

//===================Release all LTUs used by the route
FOR L_uiIndex := 1 TO Ref_stRoute.iuStepCount 
	DO
    CASE Ref_stRoute.astSteps[L_uiIndex].eConvoyer 
			OF
        E_Convoyer.Convoyer_3:  itfLTU3.ReservedBy  := E_Convoyer.Convoyer_NONE;
        E_Convoyer.Convoyer_6:  itfLTU6.ReservedBy  := E_Convoyer.Convoyer_NONE;
        E_Convoyer.Convoyer_9:  itfLTU9.ReservedBy  := E_Convoyer.Convoyer_NONE;
        E_Convoyer.Convoyer_12: itfLTU12.ReservedBy := E_Convoyer.Convoyer_NONE;
    END_CASE
END_FOR
mReleaseResources := TRUE;
END_METHOD

METHOD mReleaseRoute : E_CmdState
VAR_INPUT
	I_uiJobID					 : UINT;
END_VAR

VAR
    L_uiIndex : UINT;
END_VAR

//=================== Search job by ID and clear job
FOR L_uiIndex := 1 TO 10 DO
	IF astRouteQueue[L_uiIndex].bValid
	   AND astRouteQueue[L_uiIndex].uiJobID = I_uiJobID 
		 	THEN
				//===================Release reserved LTU resources
	  		mReleaseResources(astRouteQueue[L_uiIndex].stRoute);  
				//=================== Clear queue slot
	  		astRouteQueue[L_uiIndex].bValid     := FALSE;
	  		astRouteQueue[L_uiIndex].bReserved  := FALSE;
	  		astRouteQueue[L_uiIndex].bExecuting := FALSE;
	  		astRouteQueue[L_uiIndex].bDone      := TRUE;
	  		astRouteQueue[L_uiIndex].bError     := FALSE;
	  		mReleaseRoute := E_CmdState.Succeeded;
	  		RETURN;
	END_IF
END_FOR

mReleaseRoute := E_CmdState.NotReady;
END_METHOD

METHOD mRequestRoute : E_CmdState
VAR_INPUT
   I_bExecute     		: BOOL;
   I_eSource      		: E_Convoyer;
   I_eDestination 		: E_Convoyer;
END_VAR

VAR
	L_uiIndex						: UINT;
END_VAR
// No command requested.
IF NOT I_bExecute 
	THEN
  	mRequestRoute  		:= E_CmdState.Idle;
    RETURN;         		
END_IF              		

//======================= Invalid source or destination
IF I_eSource = E_Convoyer.Convoyer_NONE OR 
	 I_eDestination = E_Convoyer.Convoyer_NONE 
	 	THEN
    	mRequestRoute     := E_CmdState.Error;
    	RETURN;
END_IF

//======================= Search free queue slot
FOR L_uiIndex := 1 TO 10 DO
	IF NOT astRouteQueue[L_uiIndex].bValid 
		THEN
			//======================= Create new job
    	astRouteQueue[L_uiIndex].uiJobID       := uiNextJobID;
    	astRouteQueue[L_uiIndex].eSource       := I_eSource;
    	astRouteQueue[L_uiIndex].eDestination  := I_eDestination;
    	
    	astRouteQueue[L_uiIndex].bValid        := TRUE;
    	astRouteQueue[L_uiIndex].bReserved     := FALSE;
    	astRouteQueue[L_uiIndex].bExecuting    := FALSE;
    	astRouteQueue[L_uiIndex].bDone         := FALSE;
    	astRouteQueue[L_uiIndex].bError        := FALSE;

	//=======================Build route steps
	IF NOT mBuildRoute(I_eSource, I_eDestination, astRouteQueue[L_uiIndex].stRoute) 
  	THEN
    astRouteQueue[L_uiIndex].bValid := FALSE;
    mRequestRoute := E_CmdState.Error;
    RETURN;
  END_IF
  //=======================Check resources
  IF NOT mCheckRouteFree(astRouteQueue[L_uiIndex].stRoute ) 
  	THEN
    	astRouteQueue[L_uiIndex].bValid := FALSE;
    	mRequestRoute := E_CmdState.NotReady;
    	RETURN;
  END_IF
	//======================= Reserve resources. 
  IF NOT mReserveRoute(astRouteQueue[L_uiIndex].stRoute, I_eSource) 
		THEN
    	astRouteQueue[L_uiIndex].bValid := FALSE;
    	mRequestRoute := E_CmdState.NotReady;
    	RETURN;
  END_IF
	
  	astRouteQueue[L_uiIndex].bReserved := TRUE;
  	uiNextJobID := uiNextJobID + 1;
  	mRequestRoute := E_CmdState.Succeeded;
  	RETURN;
	END_IF
END_FOR
END_METHOD

METHOD mReserveRoute : BOOL
VAR_INPUT
	Ref_stRoute    : REFERENCE TO ST_Route;
	I_eReservedBy  : E_Convoyer;  // source
END_VAR

VAR
	L_uiIndex 		 : UINT;
END_VAR

//=================== Reserve all Ltu used by the route
FOR L_uiIndex := 1 TO Ref_stRoute.iuStepCount 
	DO
		CASE Ref_stRoute.astSteps[L_uiIndex].eConvoyer 
			OF
  			E_Convoyer.Convoyer_3: 	itfLTU3.ReservedBy  := I_eReservedBy;	
  			E_Convoyer.Convoyer_6: 	itfLTU6.ReservedBy  := I_eReservedBy;
  			E_Convoyer.Convoyer_9: 	itfLTU9.ReservedBy  := I_eReservedBy;
  	  	E_Convoyer.Convoyer_12: itfLTU12.ReservedBy := I_eReservedBy;
  	END_CASE
END_FOR
mReserveRoute := TRUE;
END_METHOD

METHOD mSequence : E_CmdState
VAR_INPUT
	I_bExecute				: BOOL;
END_VAR

VAR_INST
	L_eCmdState 		 : E_CmdState; // To Generic checks from parent state 
	
END_VAR

// Generic checks from parent
L_eCmdState := SUPER^.mSequence(I_bExecute := I_bExecute);

IF L_eCmdState <> E_CmdState.Busy 
	THEN
    mSequence := L_eCmdState;
    RETURN;
END_IF

CASE Mode OF
	E_Mode.Homing:
		mSequence := mCmdExec_BasePos();
	E_Mode.Auto:
		mSequence := mCmdExec_Auto();		
	E_Mode.Service:
		mSequence := mCmdExec_Service();		
END_CASE
END_METHOD

METHOD mService : E_CmdState
VAR_INPUT
	I_bExecute	: BOOL;
END_VAR

SUPER^.mService(I_bExecute);
END_METHOD

METHOD mStop : E_CmdState
VAR_INPUT
	I_bExecute	: BOOL;
END_VAR

SUPER^.mStop(I_bExecute);
END_METHOD

END_FUNCTION_BLOCK

// ---- 002 POUs/01 Lib/01 Device/FD_RouteExecutorDevice.TcPOU
FUNCTION_BLOCK FD_RouteExecutorDevice EXTENDS FD_Device 
VAR_INPUT
END_VAR

VAR_OUTPUT
END_VAR

VAR
	//===================== interface
 	itfLTU3  											: ITF_LTU;
 	itfLTU6  											: ITF_LTU;
 	itfLTU9  											: ITF_LTU;
 	itfLTU12 											: ITF_LTU;
          											
	itfC3    											: ITF_Convoyer;
	itfC6    											: ITF_Convoyer;
	itfC9    											: ITF_Convoyer;
	itfC12   											: ITF_Convoyer;
	
	itfRouteProvider							: ITF_RouteProvider;
	
	
	//===================== Variable
	// Ich muss Pointer verwenden, weil der RouteExecutor direkt mit dem echten Job arbeiten muss, 
  //der im RouteManager gespeichert ist.
	pstCurrentJob 								: POINTER TO ST_RouteJob; //
	
	uiCurrentStep 								: UINT; // Current route step index
	bJobActive 										: BOOL; // TRUE while executor is processing a route
	
	
	//===================== Instance

																								
END_VAR

VAR CONSTANT
	// --------------------------Base------------------
	C_SeqStep_OnBasePos_Start															: UINT :=  1; 
	C_SeqStep_OnBasePos_Error															: UINT :=  20;
	C_SeqStep_OnBasePos_Done															: UINT :=  20; 

	// --------------------------Auto Sequence------------------
	C_SeqStep_Auto_Start																	: UINT :=  1;
	C_SeqStep_Auto_Execute_GetNext_Route_Job							: UINT :=  50;
	C_SeqStep_Auto_Execute_Current_Route_Step							: UINT :=  60;
	C_SeqStep_Auto_Release_Current_Job										: UINT :=  70;
	C_SeqStep_Auto_Error																	: UINT :=  80;
	C_SeqStep_Auto_End																		: UINT :=  90;
	
END_VAR


//******* Important and necessary
SUPER^();  
//====================================
IF NOT Enable THEN RETURN; END_IF

//FB_Init ist immer implizit verfügbar und wird primär für die Initialisierung verwendet.
//Der Rückgabewert wird nicht ausgewertet. Für gezielte Einflussnahme können Sie
//die Methoden explizit deklarieren und darin mit dem Standard-Initialisierungscode 
//zusätzlichen Code bereitstellen. Sie können den Rückgabewert auswerten.
METHOD FB_Init: BOOL
VAR_INPUT    
	bInitRetains					: BOOL; 					// TRUE: Die Retain-Variablen werden initialisiert (Reset warm / Reset kalt)    
	bInCopyCode						: BOOL;  					// TRUE: Die Instanz wird danach in den Kopiercode kopiert (Online-Change)
	
	I_Name                : STRING;         //  Name
	I_ID                  : UINT;           // ID
  I_itfOwner					  : ITF_Owner;      // owner 
	
	// ITF_LTU	
	I_itfLTU3  						: ITF_LTU;        
 	I_itfLTU6  						: ITF_LTU;
 	I_itfLTU9  						: ITF_LTU;
 	I_itfLTU12 						: ITF_LTU;
	
	// ITF_Convoyer  							
	I_itfC3    						: ITF_Convoyer;
	I_itfC6    						: ITF_Convoyer;
	I_itfC9    						: ITF_Convoyer;
	I_itfC12   						: ITF_Convoyer;
	// Route Provider
	I_itfRouteProvider		: ITF_RouteProvider;
END_VAR

// chek and link LTU
IF I_itfLTU3  <>0 THEN itfLTU3  := I_itfLTU3; END_IF
IF I_itfLTU6  <>0 THEN itfLTU6  := I_itfLTU6; END_IF
IF I_itfLTU9  <>0 THEN itfLTU9  := I_itfLTU9; END_IF
IF I_itfLTU12 <>0 THEN itfLTU12 := I_itfLTU12;END_IF

// chek and link covoyer
IF I_itfC3  <>0 THEN itfC3  := I_itfC3; END_IF
IF I_itfC6  <>0 THEN itfC6  := I_itfC6; END_IF
IF I_itfC9  <>0 THEN itfC9  := I_itfC9; END_IF
IF I_itfC12 <>0 THEN itfC12 := I_itfC12;END_IF

// chek lind to Route manager
IF I_itfRouteProvider <>0 THEN itfRouteProvider := I_itfRouteProvider;END_IF
END_METHOD

METHOD mAutomatic : E_CmdState
VAR_INPUT
	I_bExecute	: BOOL;
END_VAR
SUPER^.mAutomatic(I_bExecute);
END_METHOD

METHOD mCmdExec_Auto : E_CmdState
VAR_INPUT
END_VAR
VAR
	L_eCmdState 			 : E_CmdState;
END_VAR


CASE SequenceID OF	
  //============================ Start
	C_SeqStep_Auto_Start:
		// Initialize the route executor state.
  	bJobActive       := FALSE;
  	uiCurrentStep    := 0;
  	//pstCurrentJob 	 := 0;
  	SequenceID       := C_SeqStep_Auto_Execute_GetNext_Route_Job;

	C_SeqStep_Auto_Execute_GetNext_Route_Job: // 10
  	// If no job is active, ask RouteManager for one
  	IF NOT bJobActive 
		THEN
  		L_eCmdState      := mGetNextJob();
  		CASE L_eCmdState OF
  		  	E_CmdState.Succeeded:
  		    	// A job was received // Start executing route steps
  		     	SequenceID := C_SeqStep_Auto_Execute_Current_Route_Step;
  		    E_CmdState.Idle:
  		    	// No job available // Stay waiting // End Auto Sequency
  		  		SequenceID := C_SeqStep_Auto_End;
  		  ELSE
  		    // Route provider error or not ready
  		  	SequenceID 	 := C_SeqStep_Error;
  			END_CASE
  		ELSE
  		  // A job is already active
  			SequenceID   	 := C_SeqStep_Auto_Execute_Current_Route_Step;
  		END_IF
			mCmdExec_Auto    := E_CmdState.Busy;
 
	C_SeqStep_Auto_Execute_Current_Route_Step: // 20
  	L_eCmdState := mExecuteCurrentStep();
    	CASE L_eCmdState OF
    	 E_CmdState.Succeeded:
    	   // If all route steps are done, release the job.
    	   IF pstCurrentJob <> 0 
				 	 THEN
    	     	 IF uiCurrentStep > pstCurrentJob^.stRoute.iuStepCount 
						   THEN
    	     	     SequenceID := C_SeqStep_Auto_Release_Current_Job;
    	     	 ELSE
    	     	   // Continue with next step.
    	     	   SequenceID := C_SeqStep_Auto_Execute_Current_Route_Step;
    	     	 END_IF
    	   ELSE
    	   	SequenceID := C_SeqStep_Error;
    	   END_IF
    	 E_CmdState.Busy:
    	   // Current step is still running
    	   SequenceID := C_SeqStep_Auto_Execute_Current_Route_Step;
    	 ELSE
    		// Any other state is considered an execution error
    		IF pstCurrentJob <> 0 THEN pstCurrentJob^.bError := TRUE; END_IF
    		SequenceID := C_SeqStep_Error;
    	END_CASE

    	mCmdExec_Auto := E_CmdState.Busy;
    	RETURN;
	
	C_SeqStep_Auto_Release_Current_Job: // 30
		L_eCmdState := mRealeaseCurrentJob();
     	CASE L_eCmdState OF
     	    E_CmdState.Succeeded:
     	    	// Job released ==> Go back and wait for next job
     	    	SequenceID := C_SeqStep_Auto_End;
     	    E_CmdState.Busy:
     	   	  // Release still running
     	   	  SequenceID := C_SeqStep_Auto_Release_Current_Job;  	  
     	    ELSE
     	      // Release failed.
     	      SequenceID := C_SeqStep_Error;  	
     	END_CASE
     	mCmdExec_Auto := E_CmdState.Busy;
     	RETURN;	
 	C_SeqStep_Auto_End:
  	SequenceID 			:= C_SeqStep_Auto_Start;
		
END_CASE
END_METHOD

METHOD mCmdExec_BasePos : E_CmdState
VAR_INPUT
END_VAR

CASE SequenceID OF
  //******************************************************* Idle 
  C_SeqStep_Idle: 
  	SequenceID       :=  C_SeqStep_OnBasePos_Start;
		
  //****************************************************** Start
  C_SeqStep_OnBasePos_Start:
	// Home position for LTU is MIDDLE.
		Homed 					 := TRUE;
  	Ready 					 := TRUE;
  	SequenceID 			 := C_SeqStep_OnBasePos_Done;
	
  C_SeqStep_Error: 
    //************* all FB reset
    mCmdExec_BasePos := mDone(); 
  //**********************Done
 	C_SeqStep_OnBasePos_Done:
  	mCmdExec_BasePos := mDone();
END_CASE
END_METHOD

METHOD mCmdExec_Service : E_CmdState
VAR_INPUT
END_VAR

 Ready 								:= TRUE;
 SequenceBusy 				:= FALSE;
 SequenceDone 				:= TRUE;
 SequenceID 					:= C_SeqStep_Idle;
 mCmdExec_Service 		:= E_CmdState.Succeeded;
 RETURN;
END_METHOD

METHOD mExecuteCurrentStep : E_CmdState
VAR_INPUT
END_VAR
VAR
	L_stStep     : ST_RouteStep;
	L_itfLTU     : ITF_LTU;
	L_eCmdState  : E_CmdState;
END_VAR

//Execute the current routing step (MoveTop, MoveBottom, transport, etc.)
// Check current job pointer
IF pstCurrentJob = 0 
	THEN
  	mExecuteCurrentStep := E_CmdState.NotReady;
    RETURN;
END_IF

// Check current step index
IF uiCurrentStep = 0 
	THEN
    mExecuteCurrentStep := E_CmdState.NotReady;
    RETURN;
END_IF

IF uiCurrentStep > pstCurrentJob^.stRoute.iuStepCount 
	THEN
    mExecuteCurrentStep := E_CmdState.Succeeded;
    RETURN;
END_IF

// Get current route step
L_stStep := pstCurrentJob^.stRoute.astSteps[uiCurrentStep];

// Get LTU linked to this convoyer
L_eCmdState := mGetLTUByConvoyer(L_stStep.eConvoyer, O_itfLTU => L_itfLTU);

IF L_eCmdState <> E_CmdState.Succeeded THEN
    mExecuteCurrentStep := L_eCmdState;
    RETURN;
END_IF

// Execute requested LTU position
//==================================================
CASE L_stStep.eLTUPosition OF
  E_LTUPosition.LTU_TOP:    L_eCmdState := L_itfLTU.mCmdExec_MoveTop(TRUE);
  E_LTUPosition.LTU_BOTTOM: L_eCmdState := L_itfLTU.mCmdExec_MoveBottom(TRUE);
  E_LTUPosition.LTU_MIDDLE: L_eCmdState := L_itfLTU.mCmdExec_MoveMiddle(TRUE);
ELSE
  mExecuteCurrentStep := E_CmdState.Error;
  RETURN;
END_CASE

CASE L_eCmdState OF
	E_CmdState.Succeeded:
		// Current step completed, move to next step.
		uiCurrentStep := uiCurrentStep + 1;
	  mExecuteCurrentStep := E_CmdState.Succeeded;
	  RETURN;
		
	E_CmdState.Busy:
	// Step still running.
		mExecuteCurrentStep := E_CmdState.Busy;
		RETURN;
	ELSE
	// Any other state is considered not ready/error.
		mExecuteCurrentStep := L_eCmdState;
		RETURN;
END_CASE
END_METHOD

METHOD mGetConvoyerByID : E_CmdState
VAR_INPUT
	I_eConvoyer : E_Convoyer;
END_VAR
VAR_OUTPUT
  O_itfConvoyer : ITF_Convoyer;
END_VAR

// Return convoyer interface corresponding to ID
CASE I_eConvoyer 
	OF
    E_Convoyer.Convoyer_3: // Convoyer 3
    	O_itfConvoyer := itfC3;
    	mGetConvoyerByID := E_CmdState.Succeeded;
    	RETURN;

    E_Convoyer.Convoyer_6:  // Convoyer 6
    	O_itfConvoyer := itfC6;
    	mGetConvoyerByID := E_CmdState.Succeeded;
    	RETURN;

    E_Convoyer.Convoyer_9: // Convoyer 9
    	O_itfConvoyer := itfC9;
    	mGetConvoyerByID := E_CmdState.Succeeded;
    	RETURN;

    E_Convoyer.Convoyer_12: // Convoyer 12
    	O_itfConvoyer := itfC12;
    	mGetConvoyerByID := E_CmdState.Succeeded;
    	RETURN;

END_CASE
//Invalid convoyer
mGetConvoyerByID := E_CmdState.Error;
END_METHOD

METHOD mGetLTUByConvoyer : E_CmdState
VAR_INPUT
	I_eConvoyer : E_Convoyer;
END_VAR

VAR_OUTPUT
  O_itfLTU : ITF_LTU;
END_VAR

// Return LTU interface corresponding to convoyer ID
CASE I_eConvoyer 
	OF
    E_Convoyer.Convoyer_3: // Convoyer 3 -> LTU3
    	O_itfLTU := itfLTU3;
    	mGetLTUByConvoyer := E_CmdState.Succeeded;
    	RETURN;

    E_Convoyer.Convoyer_6: // Convoyer 6 -> LTU6
    	O_itfLTU := itfLTU6;
    	mGetLTUByConvoyer := E_CmdState.Succeeded;
    	RETURN;

    E_Convoyer.Convoyer_9: // Convoyer 9 -> LTU9
    	O_itfLTU := itfLTU9;
    	mGetLTUByConvoyer := E_CmdState.Succeeded;
    	RETURN;

    E_Convoyer.Convoyer_12: // Convoyer 12 -> LTU12
    	O_itfLTU := itfLTU12;
    	mGetLTUByConvoyer := E_CmdState.Succeeded;
    	RETURN;
END_CASE

// Invalid convoyer
mGetLTUByConvoyer := E_CmdState.Error;
END_METHOD

METHOD mGetNextJob : E_CmdState
VAR_INPUT
END_VAR
VAR
	L_eCmdState 					: E_CmdState;
END_VAR

// Request the next available ST_RouteJob from the RouteManager

// No route provider connected
IF (itfRouteProvider = 0 ) 
	THEN
  	mGetNextJob := E_CmdState.NotReady;
  	RETURN;
END_IF

// Safety check for null pointer
IF pstCurrentJob = 0 
	THEN
    mGetNextJob := E_CmdState.Error;
    RETURN;
END_IF

// Ask RouteManager for next route job
L_eCmdState := itfRouteProvider.mGetNextRoute(O_pRouteJob => pstCurrentJob);

// Check command state.
IF L_eCmdState <> E_CmdState.Succeeded 
	THEN
    mGetNextJob := L_eCmdState;
    RETURN;
END_IF

// Job successfully received
bJobActive    := TRUE;

// Start from first step
uiCurrentStep := 1;

mGetNextJob   := E_CmdState.Succeeded;
END_METHOD

METHOD mHold : E_CmdState
VAR_INPUT
	I_bExecute	: BOOL;
END_VAR

SUPER^.mHold(I_bExecute);
END_METHOD

METHOD mHome : E_CmdState
VAR_INPUT
	I_bExecute	: BOOL;
END_VAR

SUPER^.mHome(I_bExecute);
END_METHOD

METHOD mRealeaseCurrentJob : E_CmdState
VAR_INPUT
END_VAR

VAR
	L_eCmdState : E_CmdState;
END_VAR
// Notify the RouteManager that the job is complete and release the resources
// Check route provider
IF itfRouteProvider = 0 
	THEN
    mRealeaseCurrentJob := E_CmdState.NotReady;
    RETURN;
END_IF

// Check current job pointer
IF pstCurrentJob = 0 
	THEN
    mRealeaseCurrentJob := E_CmdState.NotReady;
    RETURN;
END_IF

// Tell RouteManager to release route resources
L_eCmdState := itfRouteProvider.mReleaseRoute(pstCurrentJob^.uiJobID);

// Evaluate release result
IF L_eCmdState = E_CmdState.Succeeded 
	THEN
    // Mark local executor state as free
    bJobActive 					:= FALSE;
    // Reset step counter
    uiCurrentStep 			:= 0;
    // Clear pointer to avoid using an old job
    pstCurrentJob 			:= 0;
    mRealeaseCurrentJob := E_CmdState.Succeeded;
    RETURN;
END_IF
// Release failed
mRealeaseCurrentJob := L_eCmdState;
END_METHOD

METHOD mRelease : E_CmdState
VAR_INPUT
	I_bExecute	: BOOL;
END_VAR

SUPER^.mRelease(I_bExecute);
END_METHOD

METHOD mSequence : E_CmdState
VAR_INPUT
	I_bExecute		 : BOOL;
END_VAR

VAR_INST
	L_eCmdState 	 : E_CmdState; // To Generic checks from parent state 
END_VAR

// Generic checks from parent
L_eCmdState := SUPER^.mSequence(I_bExecute := I_bExecute);

IF L_eCmdState <> E_CmdState.Busy 
	THEN
    mSequence := L_eCmdState;
    RETURN;
END_IF

CASE Mode OF
	E_Mode.Homing:
		mSequence := mCmdExec_BasePos();
	E_Mode.Auto:
		mSequence := mCmdExec_Auto();		
	E_Mode.Service:
		mSequence := mCmdExec_Service();		
END_CASE
END_METHOD

METHOD mService : E_CmdState
VAR_INPUT
	I_bExecute	: BOOL;
END_VAR

SUPER^.mService(I_bExecute);
END_METHOD

METHOD mStop : E_CmdState
VAR_INPUT
	I_bExecute	: BOOL;
END_VAR

SUPER^.mStop(I_bExecute);
END_METHOD

END_FUNCTION_BLOCK

// ---- 002 POUs/01 Lib/02 SimpleDevice/00 Template/FB_TemplateSimpleDevice.TcPOU
FUNCTION_BLOCK FB_TemplateSimpleDevice EXTENDS FB_Base
VAR_INPUT
END_VAR
VAR_OUTPUT
END_VAR
VAR
END_VAR

//FB_Init ist immer implizit verfügbar und wird primär für die Initialisierung verwendet.
//Der Rückgabewert wird nicht ausgewertet. Für gezielte Einflussnahme können Sie
//die Methoden explizit deklarieren und darin mit dem Standard-Initialisierungscode 
//zusätzlichen Code bereitstellen. Sie können den Rückgabewert auswerten.
METHOD FB_Init: BOOL
VAR_INPUT    
	bInitRetains					: BOOL; 					// TRUE: Die Retain-Variablen werden initialisiert (Reset warm / Reset kalt)    
	bInCopyCode						: BOOL;  					// TRUE: Die Instanz wird danach in den Kopiercode kopiert (Online-Change)
	
	I_Name                : STRING;         //  Name
	I_ID                  : UINT;            // ID
END_VAR
END_METHOD

END_FUNCTION_BLOCK

// ---- 002 POUs/01 Lib/02 SimpleDevice/FB_PneuCyl_3Pos.TcPOU
FUNCTION_BLOCK FB_PneuCyl_3Pos EXTENDS FB_Base
VAR_INPUT
END_VAR
VAR_OUTPUT
END_VAR
VAR
	
	fbBottomOut												: FB_Output					  (GVL_Customer.C_Name_PneuCylBottomOut,
																													 GVL_Customer.C_ID_PneuCylBottomOut
																											  	);
																														
	fbTopOut													: FB_Output					  (GVL_Customer.C_Name_PneuCylTopOut,
																													 GVL_Customer.C_ID_PneuCylTopOut
																											  	);
	
	fbBouttomIn												: FB_Input					  (GVL_Customer.C_Name_PneuCylMiddleIn,
																													 GVL_Customer.C_ID_PneuCylMiddleIn
																											  	);

	fbTopIn 													: FB_Input					  (GVL_Customer.C_Name_PneuCylMiddleIn,
																													 GVL_Customer.C_ID_PneuCylMiddleIn
																											  	);
																												
	fbMiddleIn												: FB_Input					  (GVL_Customer.C_Name_PneuCylMiddleIn,
																													 GVL_Customer.C_ID_PneuCylMiddleIn
																											  	);
																													
																													
END_VAR

//================== Must!!
SUPER^();  
IF NOT Enable THEN RETURN; END_IF;

//FB_Init ist immer implizit verfügbar und wird primär für die Initialisierung verwendet.
//Der Rückgabewert wird nicht ausgewertet. Für gezielte Einflussnahme können Sie
//die Methoden explizit deklarieren und darin mit dem Standard-Initialisierungscode 
//zusätzlichen Code bereitstellen. Sie können den Rückgabewert auswerten.
METHOD FB_Init: BOOL
VAR_INPUT    
	bInitRetains					: BOOL; 					// TRUE: Die Retain-Variablen werden initialisiert (Reset warm / Reset kalt)    
	bInCopyCode						: BOOL;  					// TRUE: Die Instanz wird danach in den Kopiercode kopiert (Online-Change)
	
	I_Name                : STRING;         //  Name
	I_ID                  : UINT;            // ID
END_VAR
END_METHOD

METHOD mCallBottom : E_CmdState
VAR_INPUT
	I_bExecute			 : BOOL;
END_VAR
// No command requested.
IF NOT I_bExecute 
	THEN
    mCallBottom  := E_CmdState.Idle;
    RETURN;
END_IF

// Command cylinder to top.
// To Bottom=True, To Top=False.

fbBottomOut.bBoolValue 	:= TRUE;
fbTopOut.bBoolValue   	:= FALSE;

// Wait until top sensor is active.
IF fbBouttomIn.bBoolValue 
	THEN
		mCallBottom 	:= E_CmdState.Succeeded;
ELSE
    mCallBottom 	:= E_CmdState.Busy;
END_IF
END_METHOD

METHOD mCallMiddle : E_CmdState
VAR_INPUT
	I_bExecute			 : BOOL;
END_VAR
// No command requested.
IF NOT I_bExecute 
	THEN
    mCallMiddle    := E_CmdState.Idle;
    RETURN;
END_IF

// Command cylinder to Middle.
// To Bottom=False, To Top=False.
fbBottomOut.bBoolValue 	   := FALSE;
fbTopOut.bBoolValue    		 := FALSE;

// Wait until top sensor is active.
IF fbMiddleIn.bIAT_bHardwareLink 
	THEN
		mCallMiddle 	 := E_CmdState.Succeeded;
ELSE
    mCallMiddle 	 := E_CmdState.Busy;
END_IF
END_METHOD

